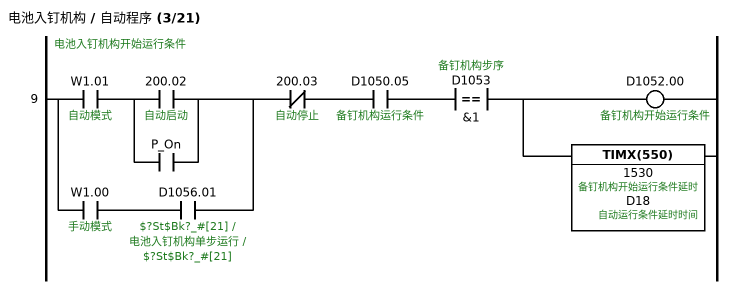
; [picture p96: 电池入钉机构 / 自动程序, rungs 9-9]
; rung 9: 电池入钉机构开始运行条件
LD W1.01  ; 自动模式
LD 200.02  ; 自动启动
OR P_On
ANDLD
LD W1.00  ; 手动模式
AND D1056.01  ; $?St$Bk?_#[21] / 电池入钉机构单步运行 / $?St$Bk?_#[21]
ORLD
ANDNOT 200.03  ; 自动停止
AND D1050.05  ; 备钉机构运行条件
AND=(300) D1053 &1  ; 备钉机构步序
OUT D1052.00  ; 备钉机构开始运行条件
TIMX(550) 1530 D18  ; 自动运行条件延时时间, 备钉机构开始运行条件延时

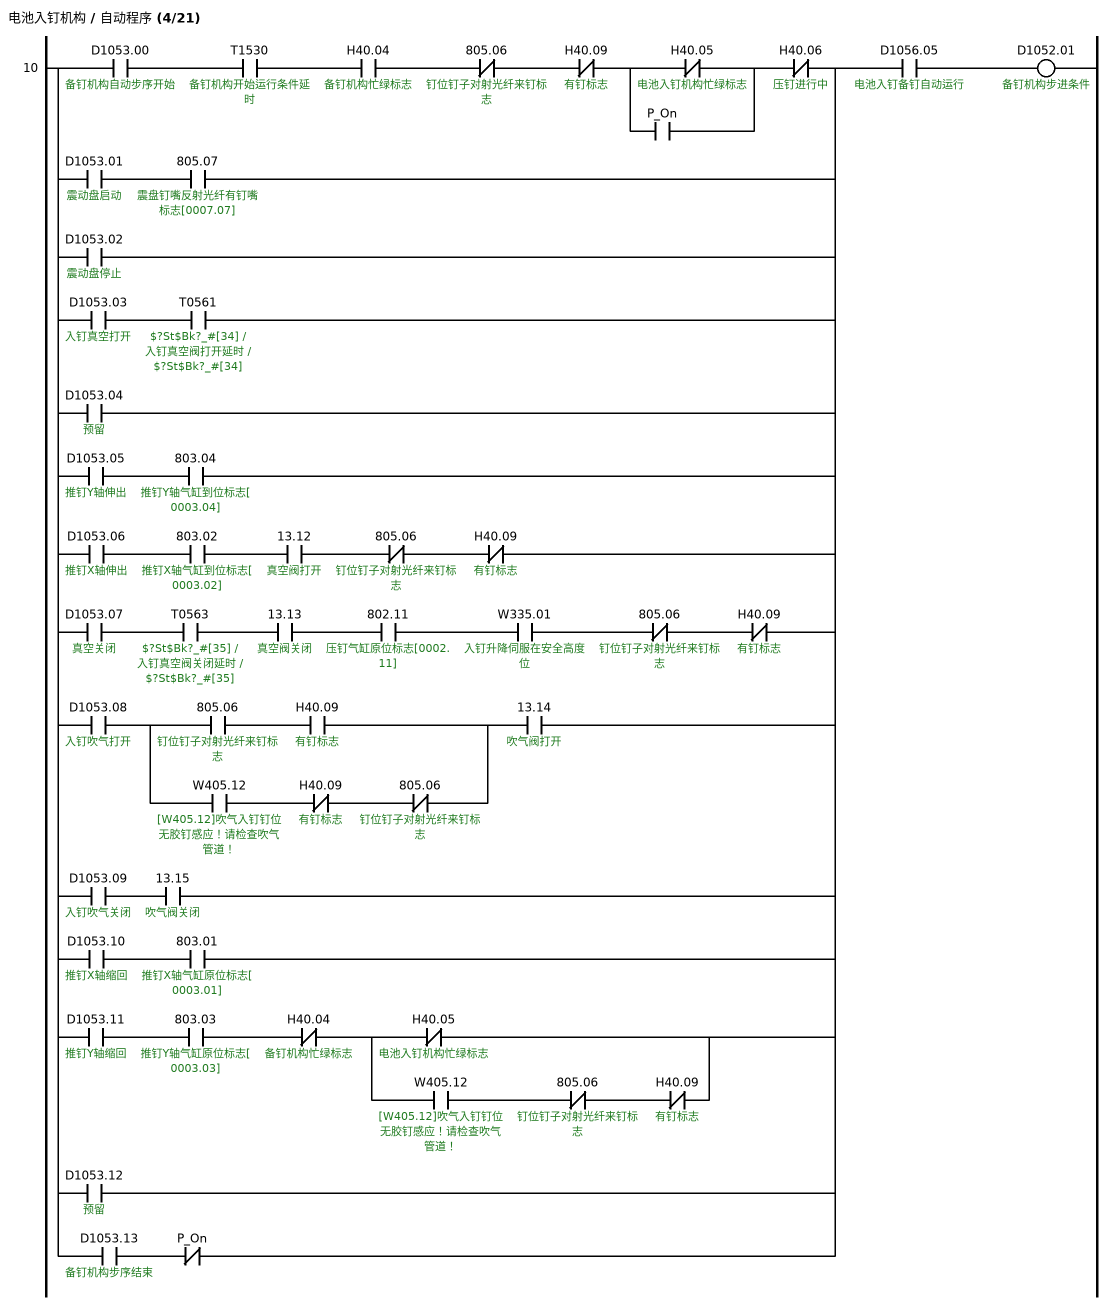
; rung 10
LD D1053.00  ; 备钉机构自动步序开始
AND T1530  ; 备钉机构开始运行条件延时
AND H40.04  ; 备钉机构忙绿标志
ANDNOT 805.06  ; 钉位钉子对射光纤来钉标志
ANDNOT H40.09  ; 有钉标志
LDNOT H40.05  ; 电池入钉机构忙绿标志
OR P_On
ANDLD
ANDNOT H40.06  ; 压钉进行中
LD D1053.01  ; 震动盘启动
AND 805.07  ; 震盘钉嘴反射光纤有钉嘴标志[0007.07]
ORLD
OR D1053.02  ; 震动盘停止
LD D1053.03  ; 入钉真空打开
AND T0561  ; $?St$Bk?_#[34] / 入钉真空阀打开延时 / $?St$Bk?_#[34]
ORLD
OR D1053.04  ; 预留
LD D1053.05  ; 推钉Y轴伸出
AND 803.04  ; 推钉Y轴气缸到位标志[0003.04]
ORLD
LD D1053.06  ; 推钉X轴伸出
AND 803.02  ; 推钉X轴气缸到位标志[0003.02]
AND 13.12  ; 真空阀打开
ANDNOT 805.06  ; 钉位钉子对射光纤来钉标志
ANDNOT H40.09  ; 有钉标志
ORLD
LD D1053.07  ; 真空关闭
AND T0563  ; $?St$Bk?_#[35] / 入钉真空阀关闭延时 / $?St$Bk?_#[35]
AND 13.13  ; 真空阀关闭
AND 802.11  ; 压钉气缸原位标志[0002.11]
AND W335.01  ; 入钉升降伺服在安全高度位
ANDNOT 805.06  ; 钉位钉子对射光纤来钉标志
ANDNOT H40.09  ; 有钉标志
ORLD
LD D1053.08  ; 入钉吹气打开
LD 805.06  ; 钉位钉子对射光纤来钉标志
AND H40.09  ; 有钉标志
LD W405.12  ; [W405.12]吹气入钉钉位无胶钉感应！请检查吹气管道！
ANDNOT H40.09  ; 有钉标志
ANDNOT 805.06  ; 钉位钉子对射光纤来钉标志
ORLD
ANDLD
AND 13.14  ; 吹气阀打开
ORLD
LD D1053.09  ; 入钉吹气关闭
AND 13.15  ; 吹气阀关闭
ORLD
LD D1053.10  ; 推钉X轴缩回
AND 803.01  ; 推钉X轴气缸原位标志[0003.01]
ORLD
LD D1053.11  ; 推钉Y轴缩回
AND 803.03  ; 推钉Y轴气缸原位标志[0003.03]
ANDNOT H40.04  ; 备钉机构忙绿标志
LDNOT H40.05  ; 电池入钉机构忙绿标志
LD W405.12  ; [W405.12]吹气入钉钉位无胶钉感应！请检查吹气管道！
ANDNOT 805.06  ; 钉位钉子对射光纤来钉标志
ANDNOT H40.09  ; 有钉标志
ORLD
ANDLD
ORLD
OR D1053.12  ; 预留
LD D1053.13  ; 备钉机构步序结束
ANDNOT P_On
ORLD
AND D1056.05  ; 电池入钉备钉自动运行
OUT D1052.01  ; 备钉机构步进条件

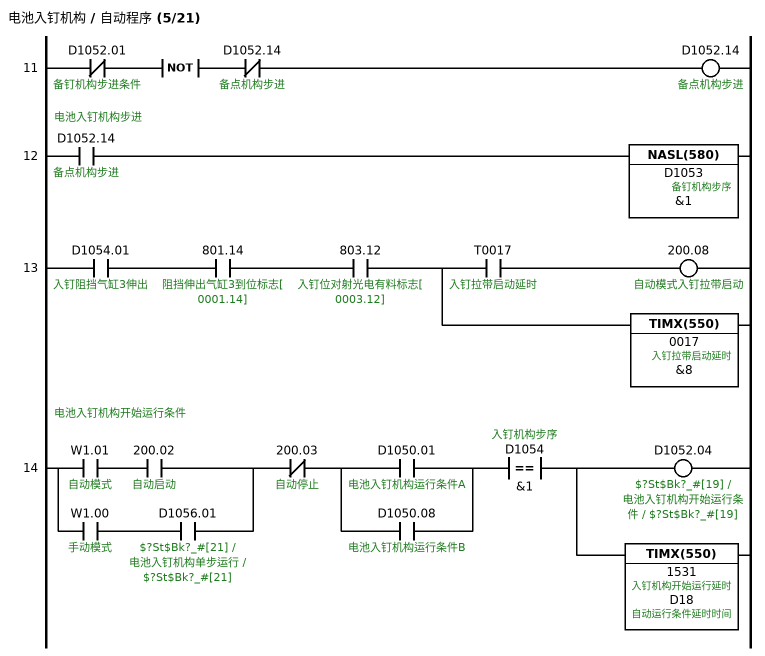
; rung 11
LDNOT D1052.01  ; 备钉机构步进条件
NOT(520)
ANDNOT D1052.14  ; 备点机构步进
OUT D1052.14  ; 备点机构步进
; rung 12: 电池入钉机构步进
LD D1052.14  ; 备点机构步进
NASL(580) D1053 &1  ; 备钉机构步序
; rung 13
LD D1054.01  ; 入钉阻挡气缸3伸出
AND 801.14  ; 阻挡伸出气缸3到位标志[0001.14]
AND 803.12  ; 入钉位对射光电有料标志[0003.12]
OUT TR0
AND T0017  ; 入钉拉带启动延时
OUT 200.08  ; 自动模式入钉拉带启动
LD TR0
TIMX(550) 0017 &8  ; 入钉拉带启动延时
; rung 14: 电池入钉机构开始运行条件
LD W1.01  ; 自动模式
AND 200.02  ; 自动启动
LD W1.00  ; 手动模式
AND D1056.01  ; $?St$Bk?_#[21] / 电池入钉机构单步运行 / $?St$Bk?_#[21]
ORLD
ANDNOT 200.03  ; 自动停止
LD D1050.01  ; 电池入钉机构运行条件A
OR D1050.08  ; 电池入钉机构运行条件B
ANDLD
AND=(300) D1054 &1  ; 入钉机构步序
OUT D1052.04  ; $?St$Bk?_#[19] / 电池入钉机构开始运行条件 / $?St$Bk?_#[19]
TIMX(550) 1531 D18  ; 自动运行条件延时时间, 入钉机构开始运行延时

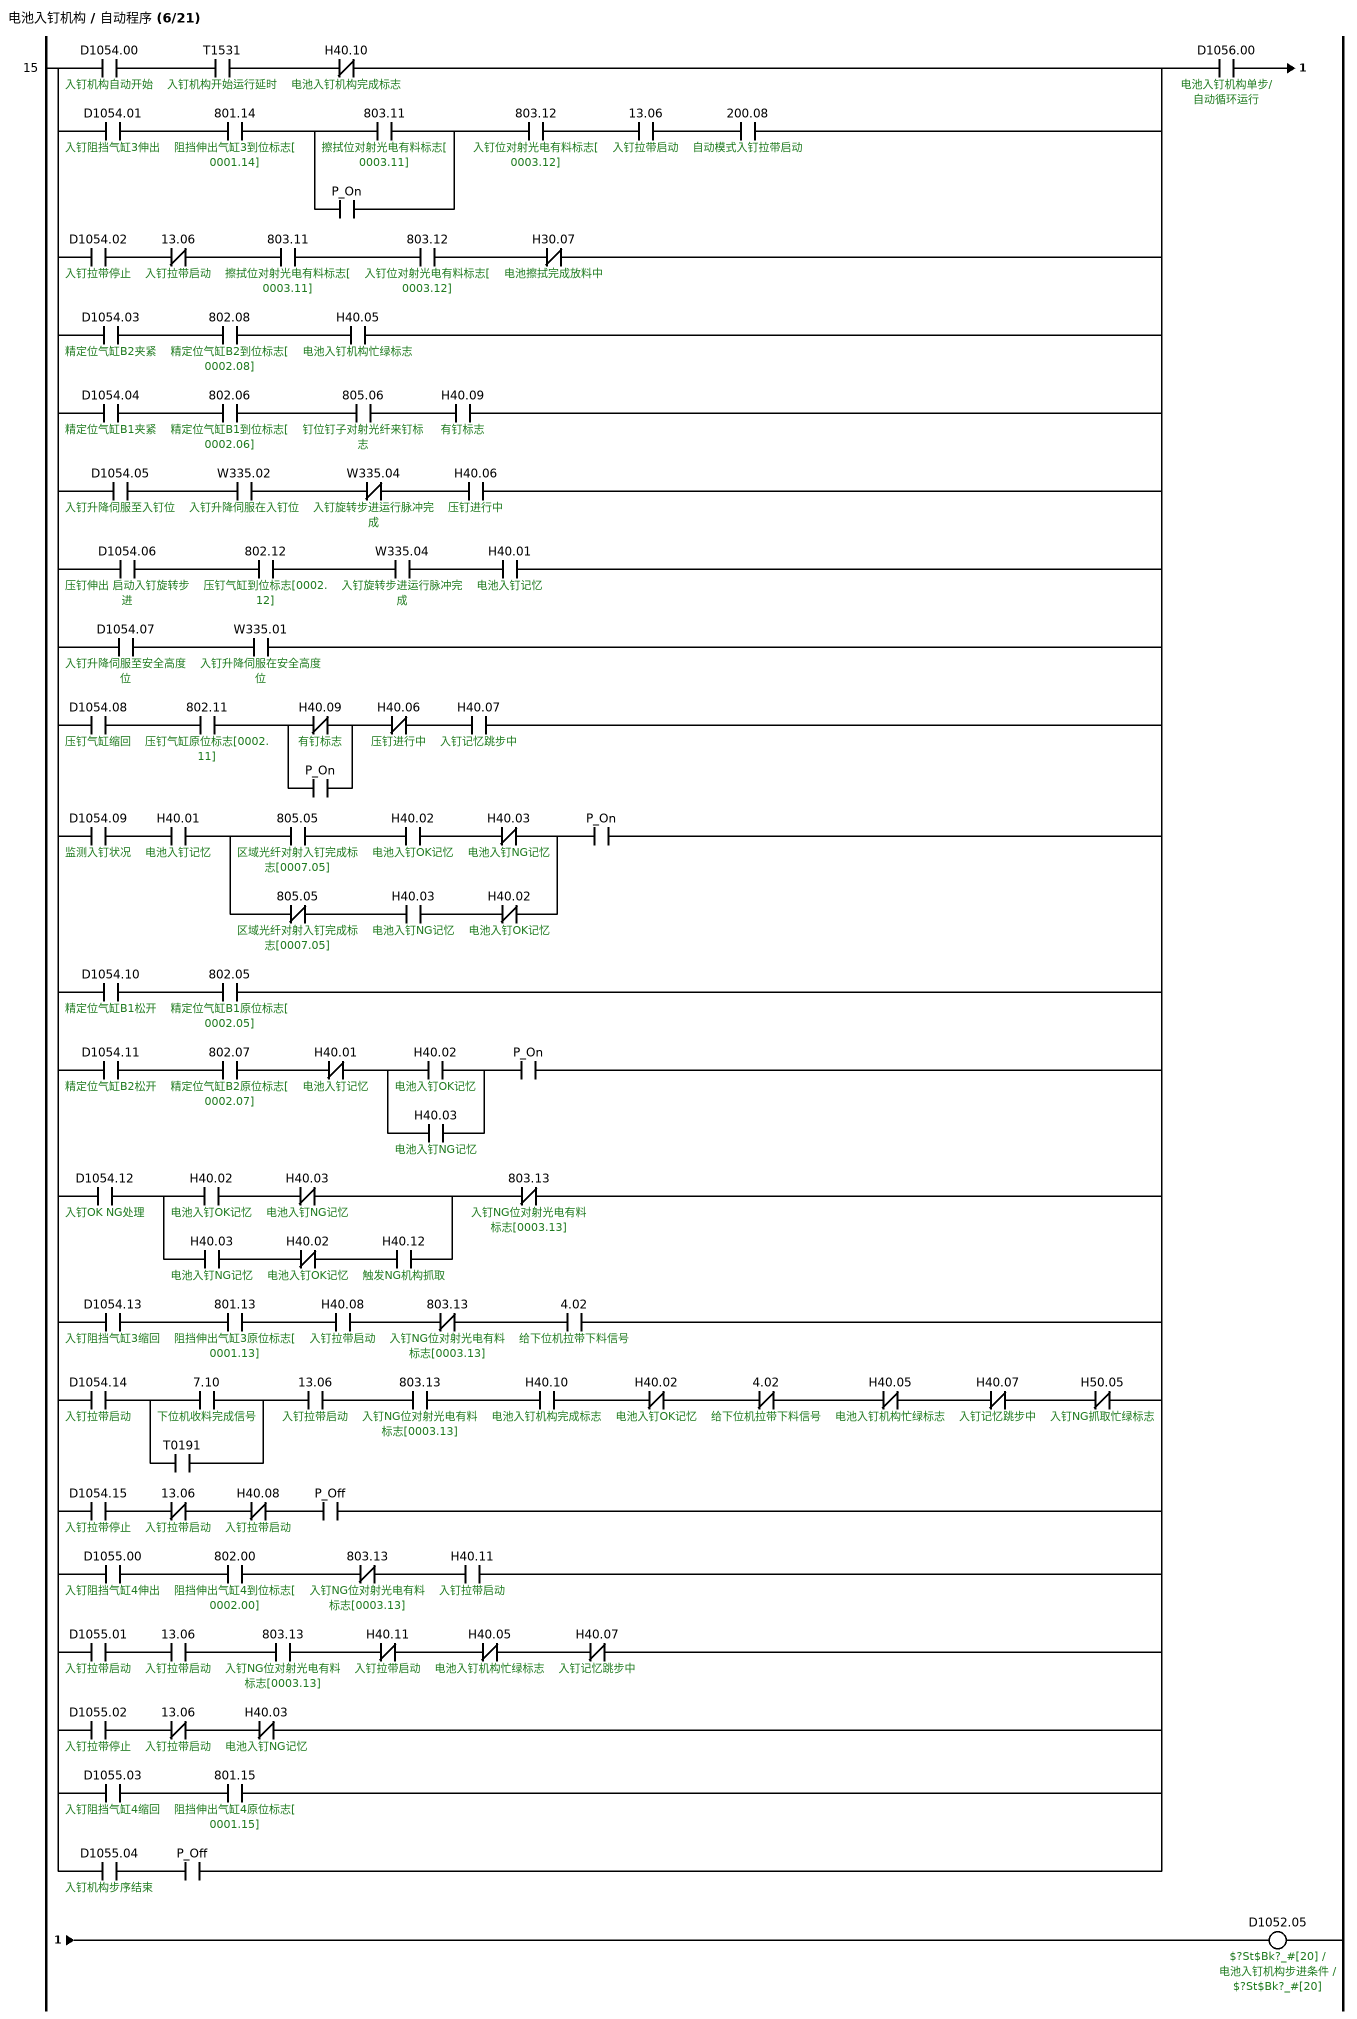
; rung 15
LD D1054.00  ; 入钉机构自动开始
AND T1531  ; 入钉机构开始运行延时
ANDNOT H40.10  ; 电池入钉机构完成标志
LD D1054.01  ; 入钉阻挡气缸3伸出
AND 801.14  ; 阻挡伸出气缸3到位标志[0001.14]
LD 803.11  ; 擦拭位对射光电有料标志[0003.11]
OR P_On
ANDLD
AND 803.12  ; 入钉位对射光电有料标志[0003.12]
AND 13.06  ; 入钉拉带启动
AND 200.08  ; 自动模式入钉拉带启动
ORLD
LD D1054.02  ; 入钉拉带停止
ANDNOT 13.06  ; 入钉拉带启动
AND 803.11  ; 擦拭位对射光电有料标志[0003.11]
AND 803.12  ; 入钉位对射光电有料标志[0003.12]
ANDNOT H30.07  ; 电池擦拭完成放料中
ORLD
LD D1054.03  ; 精定位气缸B2夹紧
AND 802.08  ; 精定位气缸B2到位标志[0002.08]
AND H40.05  ; 电池入钉机构忙绿标志
ORLD
LD D1054.04  ; 精定位气缸B1夹紧
AND 802.06  ; 精定位气缸B1到位标志[0002.06]
AND 805.06  ; 钉位钉子对射光纤来钉标志
AND H40.09  ; 有钉标志
ORLD
LD D1054.05  ; 入钉升降伺服至入钉位
AND W335.02  ; 入钉升降伺服在入钉位
ANDNOT W335.04  ; 入钉旋转步进运行脉冲完成
AND H40.06  ; 压钉进行中
ORLD
LD D1054.06  ; 压钉伸出 启动入钉旋转步进
AND 802.12  ; 压钉气缸到位标志[0002.12]
AND W335.04  ; 入钉旋转步进运行脉冲完成
AND H40.01  ; 电池入钉记忆
ORLD
LD D1054.07  ; 入钉升降伺服至安全高度位
AND W335.01  ; 入钉升降伺服在安全高度位
ORLD
LD D1054.08  ; 压钉气缸缩回
AND 802.11  ; 压钉气缸原位标志[0002.11]
LDNOT H40.09  ; 有钉标志
OR P_On
ANDLD
ANDNOT H40.06  ; 压钉进行中
AND H40.07  ; 入钉记忆跳步中
ORLD
LD D1054.09  ; 监测入钉状况
AND H40.01  ; 电池入钉记忆
LD 805.05  ; 区域光纤对射入钉完成标志[0007.05]
AND H40.02  ; 电池入钉OK记忆
ANDNOT H40.03  ; 电池入钉NG记忆
LDNOT 805.05  ; 区域光纤对射入钉完成标志[0007.05]
AND H40.03  ; 电池入钉NG记忆
ANDNOT H40.02  ; 电池入钉OK记忆
ORLD
ANDLD
AND P_On
ORLD
LD D1054.10  ; 精定位气缸B1松开
AND 802.05  ; 精定位气缸B1原位标志[0002.05]
ORLD
LD D1054.11  ; 精定位气缸B2松开
AND 802.07  ; 精定位气缸B2原位标志[0002.07]
ANDNOT H40.01  ; 电池入钉记忆
LD H40.02  ; 电池入钉OK记忆
OR H40.03  ; 电池入钉NG记忆
ANDLD
AND P_On
ORLD
LD D1054.12  ; 入钉OK NG处理
LD H40.02  ; 电池入钉OK记忆
ANDNOT H40.03  ; 电池入钉NG记忆
LD H40.03  ; 电池入钉NG记忆
ANDNOT H40.02  ; 电池入钉OK记忆
AND H40.12  ; 触发NG机构抓取
ORLD
ANDLD
ANDNOT 803.13  ; 入钉NG位对射光电有料标志[0003.13]
ORLD
LD D1054.13  ; 入钉阻挡气缸3缩回
AND 801.13  ; 阻挡伸出气缸3原位标志[0001.13]
AND H40.08  ; 入钉拉带启动
ANDNOT 803.13  ; 入钉NG位对射光电有料标志[0003.13]
AND 4.02  ; 给下位机拉带下料信号
ORLD
LD D1054.14  ; 入钉拉带启动
LD 7.10  ; 下位机收料完成信号
OR T0191
ANDLD
AND 13.06  ; 入钉拉带启动
AND 803.13  ; 入钉NG位对射光电有料标志[0003.13]
AND H40.10  ; 电池入钉机构完成标志
ANDNOT H40.02  ; 电池入钉OK记忆
ANDNOT 4.02  ; 给下位机拉带下料信号
ANDNOT H40.05  ; 电池入钉机构忙绿标志
ANDNOT H40.07  ; 入钉记忆跳步中
ANDNOT H50.05  ; 入钉NG抓取忙绿标志
ORLD
LD D1054.15  ; 入钉拉带停止
ANDNOT 13.06  ; 入钉拉带启动
ANDNOT H40.08  ; 入钉拉带启动
AND P_Off
ORLD
LD D1055.00  ; 入钉阻挡气缸4伸出
AND 802.00  ; 阻挡伸出气缸4到位标志[0002.00]
ANDNOT 803.13  ; 入钉NG位对射光电有料标志[0003.13]
AND H40.11  ; 入钉拉带启动
ORLD
LD D1055.01  ; 入钉拉带启动
AND 13.06  ; 入钉拉带启动
AND 803.13  ; 入钉NG位对射光电有料标志[0003.13]
ANDNOT H40.11  ; 入钉拉带启动
ANDNOT H40.05  ; 电池入钉机构忙绿标志
ANDNOT H40.07  ; 入钉记忆跳步中
ORLD
LD D1055.02  ; 入钉拉带停止
ANDNOT 13.06  ; 入钉拉带启动
ANDNOT H40.03  ; 电池入钉NG记忆
ORLD
LD D1055.03  ; 入钉阻挡气缸4缩回
AND 801.15  ; 阻挡伸出气缸4原位标志[0001.15]
ORLD
LD D1055.04  ; 入钉机构步序结束
AND P_Off
ORLD
AND D1056.00  ; 电池入钉机构单步/自动循环运行
OUT D1052.05  ; $?St$Bk?_#[20] / 电池入钉机构步进条件 / $?St$Bk?_#[20]

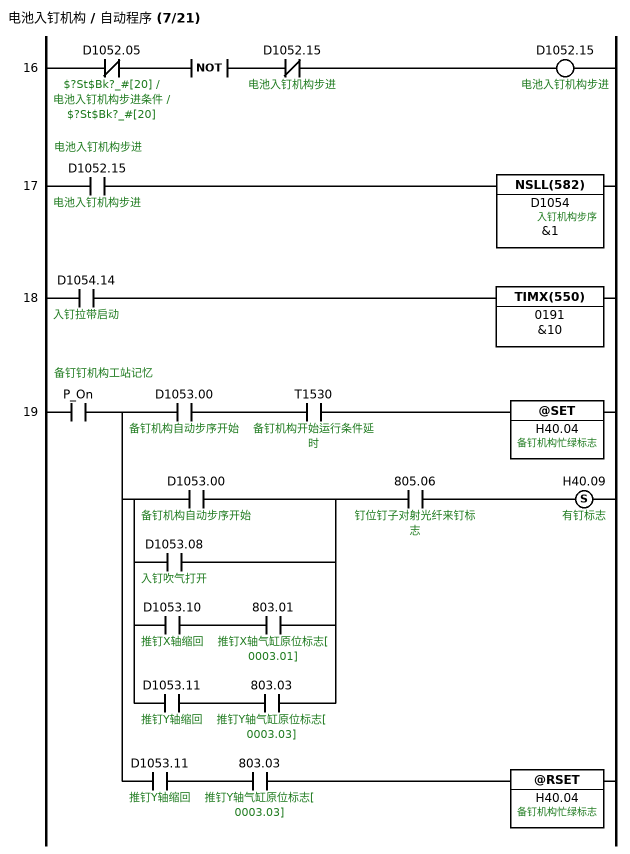
; rung 16
LDNOT D1052.05  ; $?St$Bk?_#[20] / 电池入钉机构步进条件 / $?St$Bk?_#[20]
NOT(520)
ANDNOT D1052.15  ; 电池入钉机构步进
OUT D1052.15  ; 电池入钉机构步进
; rung 17: 电池入钉机构步进
LD D1052.15  ; 电池入钉机构步进
NSLL(582) D1054 &1  ; 入钉机构步序
; rung 18
LD D1054.14  ; 入钉拉带启动
TIMX(550) 0191 &10
; rung 19: 备钉钉机构工站记忆
LD P_On
OUT TR0
AND D1053.00  ; 备钉机构自动步序开始
AND T1530  ; 备钉机构开始运行条件延时
@SET H40.04  ; 备钉机构忙绿标志
LD TR0
LD D1053.00  ; 备钉机构自动步序开始
OR D1053.08  ; 入钉吹气打开
LD D1053.10  ; 推钉X轴缩回
AND 803.01  ; 推钉X轴气缸原位标志[0003.01]
ORLD
LD D1053.11  ; 推钉Y轴缩回
AND 803.03  ; 推钉Y轴气缸原位标志[0003.03]
ORLD
ANDLD
AND 805.06  ; 钉位钉子对射光纤来钉标志
SET H40.09  ; 有钉标志
LD TR0
AND D1053.11  ; 推钉Y轴缩回
AND 803.03  ; 推钉Y轴气缸原位标志[0003.03]
@RSET H40.04  ; 备钉机构忙绿标志

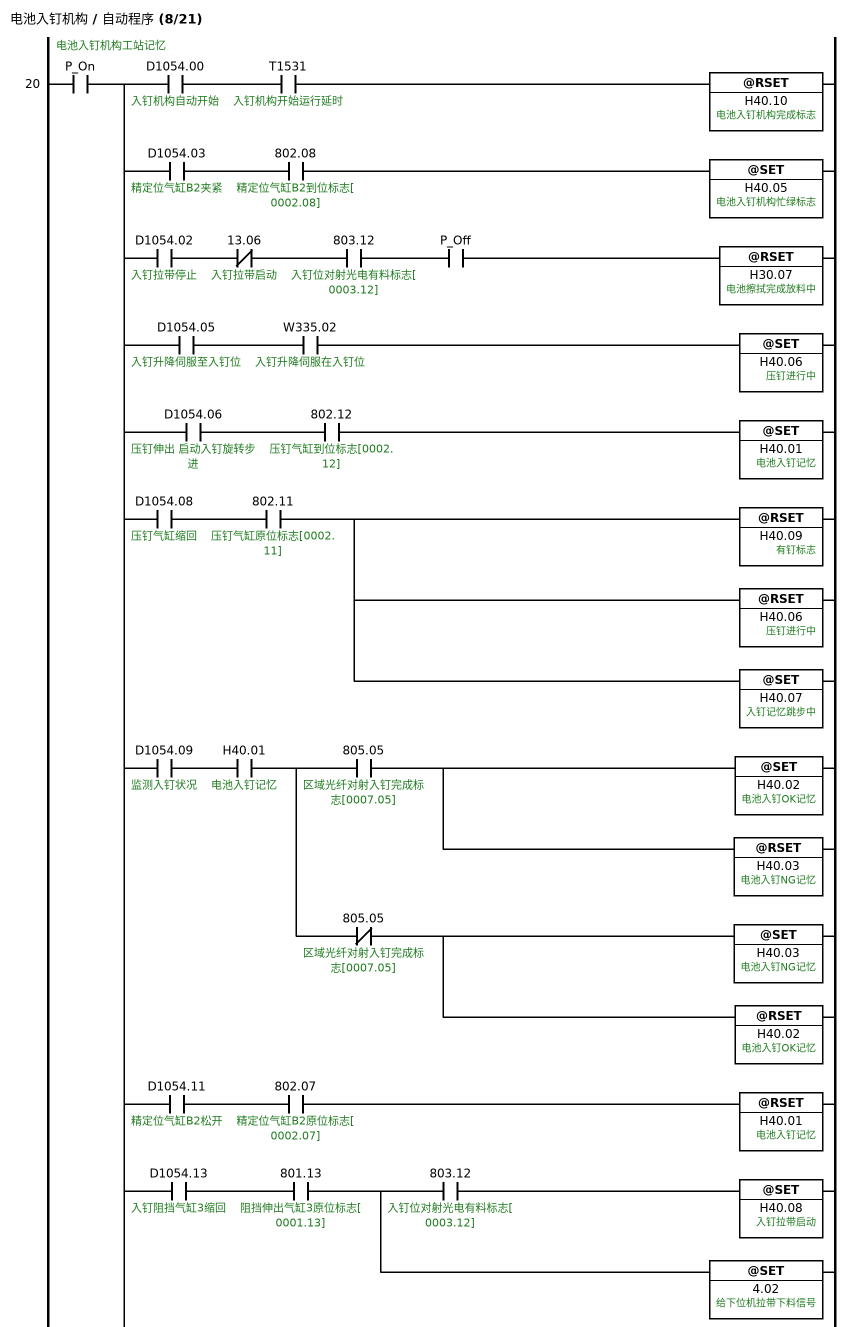

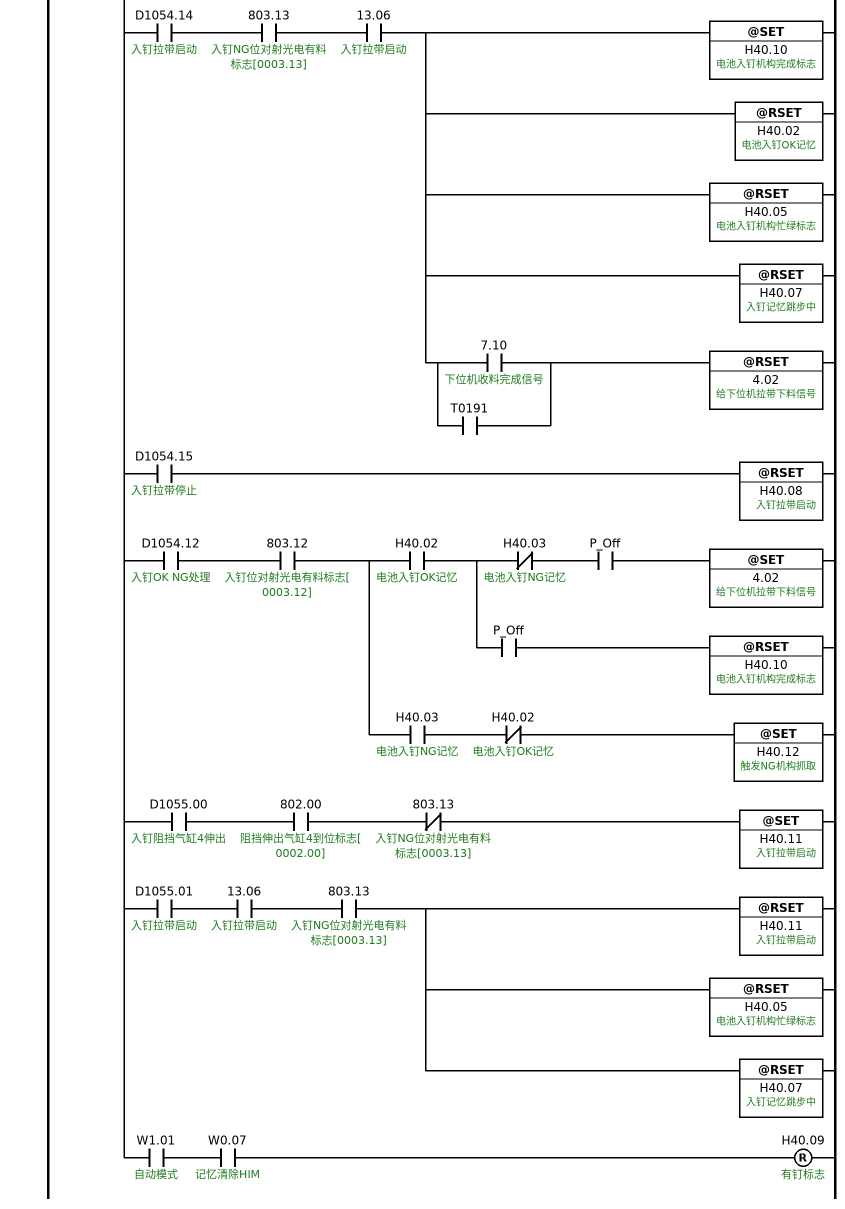
; rung 20: 电池入钉机构工站记忆
LD P_On
OUT TR0
AND D1054.00  ; 入钉机构自动开始
AND T1531  ; 入钉机构开始运行延时
@RSET H40.10  ; 电池入钉机构完成标志
LD TR0
AND D1054.03  ; 精定位气缸B2夹紧
AND 802.08  ; 精定位气缸B2到位标志[0002.08]
@SET H40.05  ; 电池入钉机构忙绿标志
LD TR0
AND D1054.02  ; 入钉拉带停止
ANDNOT 13.06  ; 入钉拉带启动
AND 803.12  ; 入钉位对射光电有料标志[0003.12]
AND P_Off
@RSET H30.07  ; 电池擦拭完成放料中
LD TR0
AND D1054.05  ; 入钉升降伺服至入钉位
AND W335.02  ; 入钉升降伺服在入钉位
@SET H40.06  ; 压钉进行中
LD TR0
AND D1054.06  ; 压钉伸出 启动入钉旋转步进
AND 802.12  ; 压钉气缸到位标志[0002.12]
@SET H40.01  ; 电池入钉记忆
LD TR0
AND D1054.08  ; 压钉气缸缩回
AND 802.11  ; 压钉气缸原位标志[0002.11]
@RSET H40.09  ; 有钉标志
@RSET H40.06  ; 压钉进行中
@SET H40.07  ; 入钉记忆跳步中
LD TR0
AND D1054.09  ; 监测入钉状况
AND H40.01  ; 电池入钉记忆
OUT TR1
AND 805.05  ; 区域光纤对射入钉完成标志[0007.05]
@SET H40.02  ; 电池入钉OK记忆
@RSET H40.03  ; 电池入钉NG记忆
LD TR1
ANDNOT 805.05  ; 区域光纤对射入钉完成标志[0007.05]
@SET H40.03  ; 电池入钉NG记忆
@RSET H40.02  ; 电池入钉OK记忆
LD TR0
AND D1054.11  ; 精定位气缸B2松开
AND 802.07  ; 精定位气缸B2原位标志[0002.07]
@RSET H40.01  ; 电池入钉记忆
LD TR0
AND D1054.13  ; 入钉阻挡气缸3缩回
AND 801.13  ; 阻挡伸出气缸3原位标志[0001.13]
OUT TR1
AND 803.12  ; 入钉位对射光电有料标志[0003.12]
@SET H40.08  ; 入钉拉带启动
LD TR1
@SET 4.02  ; 给下位机拉带下料信号
LD TR0
AND D1054.14  ; 入钉拉带启动
AND 803.13  ; 入钉NG位对射光电有料标志[0003.13]
AND 13.06  ; 入钉拉带启动
@SET H40.10  ; 电池入钉机构完成标志
@RSET H40.02  ; 电池入钉OK记忆
@RSET H40.05  ; 电池入钉机构忙绿标志
@RSET H40.07  ; 入钉记忆跳步中
LD 7.10  ; 下位机收料完成信号
OR T0191
ANDLD
@RSET 4.02  ; 给下位机拉带下料信号
LD TR0
AND D1054.15  ; 入钉拉带停止
@RSET H40.08  ; 入钉拉带启动
LD TR0
AND D1054.12  ; 入钉OK NG处理
AND 803.12  ; 入钉位对射光电有料标志[0003.12]
OUT TR1
AND H40.02  ; 电池入钉OK记忆
OUT TR2
ANDNOT H40.03  ; 电池入钉NG记忆
AND P_Off
@SET 4.02  ; 给下位机拉带下料信号
LD TR2
AND P_Off
@RSET H40.10  ; 电池入钉机构完成标志
LD TR1
AND H40.03  ; 电池入钉NG记忆
ANDNOT H40.02  ; 电池入钉OK记忆
@SET H40.12  ; 触发NG机构抓取
LD TR0
AND D1055.00  ; 入钉阻挡气缸4伸出
AND 802.00  ; 阻挡伸出气缸4到位标志[0002.00]
ANDNOT 803.13  ; 入钉NG位对射光电有料标志[0003.13]
@SET H40.11  ; 入钉拉带启动
LD TR0
AND D1055.01  ; 入钉拉带启动
AND 13.06  ; 入钉拉带启动
AND 803.13  ; 入钉NG位对射光电有料标志[0003.13]
@RSET H40.11  ; 入钉拉带启动
@RSET H40.05  ; 电池入钉机构忙绿标志
@RSET H40.07  ; 入钉记忆跳步中
LD TR0
AND W1.01  ; 自动模式
AND W0.07  ; 记忆清除HIM
RSET H40.09  ; 有钉标志

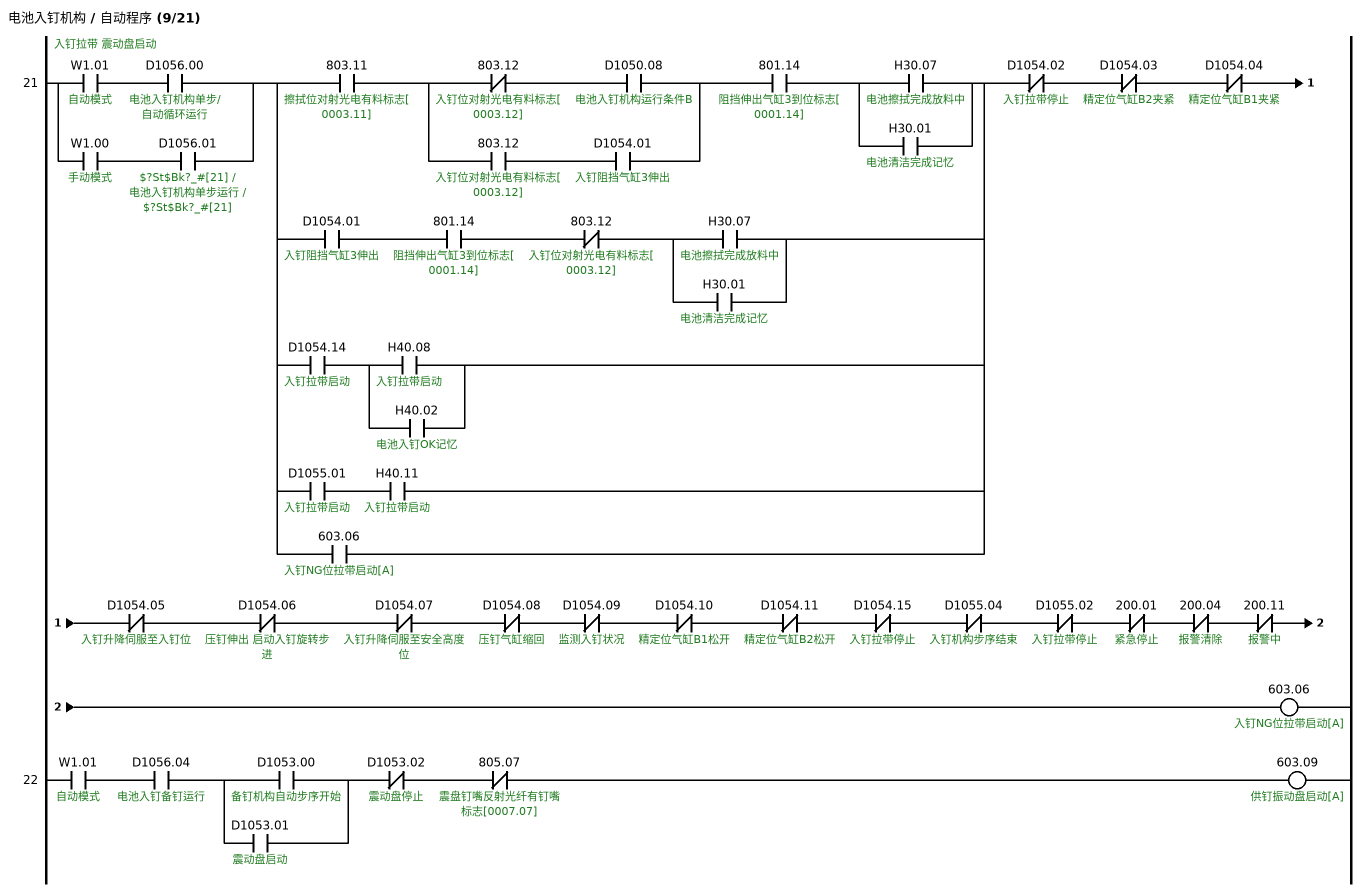
; rung 21: 入钉拉带 震动盘启动
LD W1.01  ; 自动模式
AND D1056.00  ; 电池入钉机构单步/自动循环运行
LD W1.00  ; 手动模式
AND D1056.01  ; $?St$Bk?_#[21] / 电池入钉机构单步运行 / $?St$Bk?_#[21]
ORLD
LD 803.11  ; 擦拭位对射光电有料标志[0003.11]
LDNOT 803.12  ; 入钉位对射光电有料标志[0003.12]
AND D1050.08  ; 电池入钉机构运行条件B
LD 803.12  ; 入钉位对射光电有料标志[0003.12]
AND D1054.01  ; 入钉阻挡气缸3伸出
ORLD
ANDLD
AND 801.14  ; 阻挡伸出气缸3到位标志[0001.14]
LD H30.07  ; 电池擦拭完成放料中
OR H30.01  ; 电池清洁完成记忆
ANDLD
LD D1054.01  ; 入钉阻挡气缸3伸出
AND 801.14  ; 阻挡伸出气缸3到位标志[0001.14]
ANDNOT 803.12  ; 入钉位对射光电有料标志[0003.12]
LD H30.07  ; 电池擦拭完成放料中
OR H30.01  ; 电池清洁完成记忆
ANDLD
ORLD
LD D1054.14  ; 入钉拉带启动
LD H40.08  ; 入钉拉带启动
OR H40.02  ; 电池入钉OK记忆
ANDLD
ORLD
LD D1055.01  ; 入钉拉带启动
AND H40.11  ; 入钉拉带启动
ORLD
OR 603.06  ; 入钉NG位拉带启动[A]
ANDLD
ANDNOT D1054.02  ; 入钉拉带停止
ANDNOT D1054.03  ; 精定位气缸B2夹紧
ANDNOT D1054.04  ; 精定位气缸B1夹紧
ANDNOT D1054.05  ; 入钉升降伺服至入钉位
ANDNOT D1054.06  ; 压钉伸出 启动入钉旋转步进
ANDNOT D1054.07  ; 入钉升降伺服至安全高度位
ANDNOT D1054.08  ; 压钉气缸缩回
ANDNOT D1054.09  ; 监测入钉状况
ANDNOT D1054.10  ; 精定位气缸B1松开
ANDNOT D1054.11  ; 精定位气缸B2松开
ANDNOT D1054.15  ; 入钉拉带停止
ANDNOT D1055.04  ; 入钉机构步序结束
ANDNOT D1055.02  ; 入钉拉带停止
ANDNOT 200.01  ; 紧急停止
ANDNOT 200.04  ; 报警清除
ANDNOT 200.11  ; 报警中
OUT 603.06  ; 入钉NG位拉带启动[A]
; rung 22
LD W1.01  ; 自动模式
AND D1056.04  ; 电池入钉备钉运行
LD D1053.00  ; 备钉机构自动步序开始
OR D1053.01  ; 震动盘启动
ANDLD
ANDNOT D1053.02  ; 震动盘停止
ANDNOT 805.07  ; 震盘钉嘴反射光纤有钉嘴标志[0007.07]
OUT 603.09  ; 供钉振动盘启动[A]

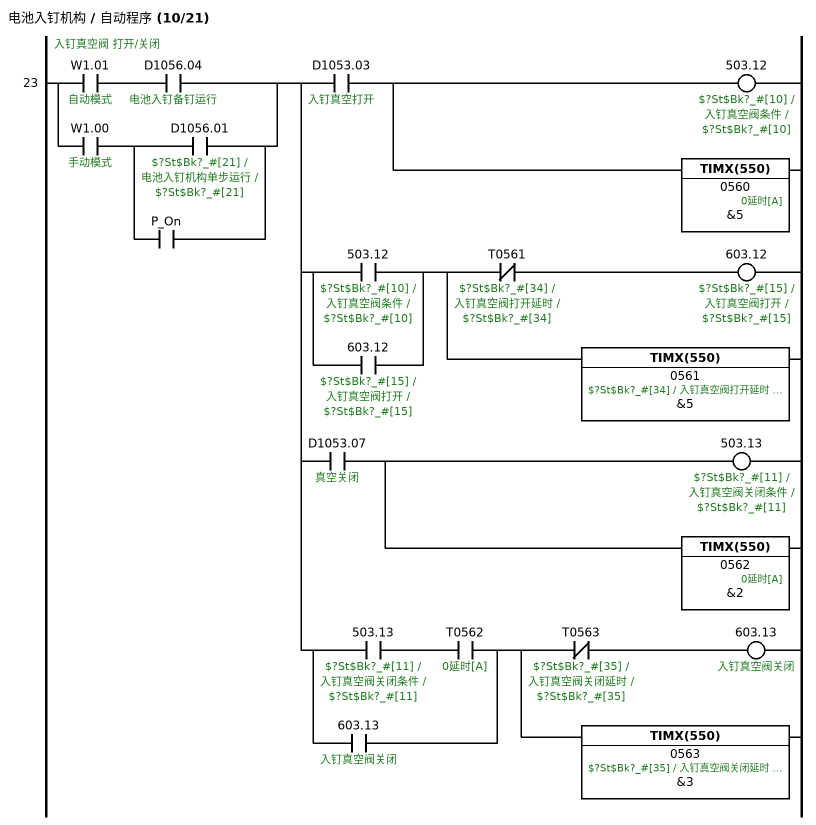
; rung 23: 入钉真空阀 打开/关闭
LD W1.01  ; 自动模式
AND D1056.04  ; 电池入钉备钉运行
LD W1.00  ; 手动模式
LD D1056.01  ; $?St$Bk?_#[21] / 电池入钉机构单步运行 / $?St$Bk?_#[21]
OR P_On
ANDLD
ORLD
OUT TR0
AND D1053.03  ; 入钉真空打开
OUT 503.12  ; $?St$Bk?_#[10] / 入钉真空阀条件 / $?St$Bk?_#[10]
TIMX(550) 0560 &5  ; 0延时[A]
LD TR0
LD 503.12  ; $?St$Bk?_#[10] / 入钉真空阀条件 / $?St$Bk?_#[10]
OR 603.12  ; $?St$Bk?_#[15] / 入钉真空阀打开 / $?St$Bk?_#[15]
ANDLD
OUT TR1
ANDNOT T0561  ; $?St$Bk?_#[34] / 入钉真空阀打开延时 / $?St$Bk?_#[34]
OUT 603.12  ; $?St$Bk?_#[15] / 入钉真空阀打开 / $?St$Bk?_#[15]
LD TR1
TIMX(550) 0561 &5  ; $?St$Bk?_#[34] / 入钉真空阀打开延时 / $?St$Bk?_#[34]
LD TR0
AND D1053.07  ; 真空关闭
OUT 503.13  ; $?St$Bk?_#[11] / 入钉真空阀关闭条件 / $?St$Bk?_#[11]
TIMX(550) 0562 &2  ; 0延时[A]
LD TR0
LD 503.13  ; $?St$Bk?_#[11] / 入钉真空阀关闭条件 / $?St$Bk?_#[11]
AND T0562  ; 0延时[A]
OR 603.13  ; 入钉真空阀关闭
ANDLD
OUT TR0
ANDNOT T0563  ; $?St$Bk?_#[35] / 入钉真空阀关闭延时 / $?St$Bk?_#[35]
OUT 603.13  ; 入钉真空阀关闭
LD TR0
TIMX(550) 0563 &3  ; $?St$Bk?_#[35] / 入钉真空阀关闭延时 / $?St$Bk?_#[35]

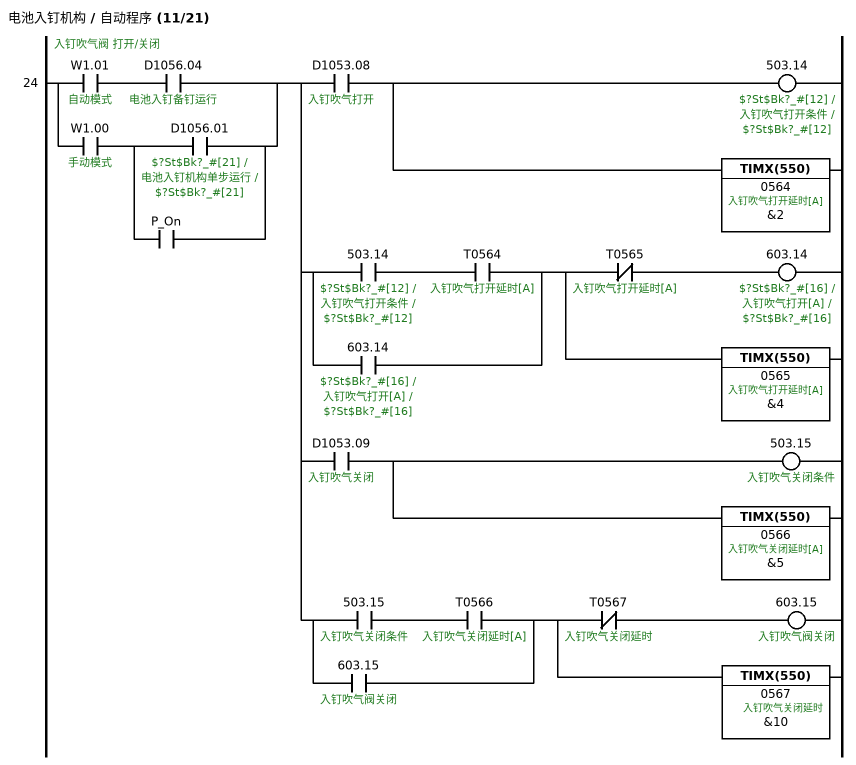
; rung 24: 入钉吹气阀 打开/关闭
LD W1.01  ; 自动模式
AND D1056.04  ; 电池入钉备钉运行
LD W1.00  ; 手动模式
LD D1056.01  ; $?St$Bk?_#[21] / 电池入钉机构单步运行 / $?St$Bk?_#[21]
OR P_On
ANDLD
ORLD
OUT TR0
AND D1053.08  ; 入钉吹气打开
OUT 503.14  ; $?St$Bk?_#[12] / 入钉吹气打开条件 / $?St$Bk?_#[12]
TIMX(550) 0564 &2  ; 入钉吹气打开延时[A]
LD TR0
LD 503.14  ; $?St$Bk?_#[12] / 入钉吹气打开条件 / $?St$Bk?_#[12]
AND T0564  ; 入钉吹气打开延时[A]
OR 603.14  ; $?St$Bk?_#[16] / 入钉吹气打开[A] / $?St$Bk?_#[16]
ANDLD
OUT TR1
ANDNOT T0565  ; 入钉吹气打开延时[A]
OUT 603.14  ; $?St$Bk?_#[16] / 入钉吹气打开[A] / $?St$Bk?_#[16]
LD TR1
TIMX(550) 0565 &4  ; 入钉吹气打开延时[A]
LD TR0
AND D1053.09  ; 入钉吹气关闭
OUT 503.15  ; 入钉吹气关闭条件
TIMX(550) 0566 &5  ; 入钉吹气关闭延时[A]
LD TR0
LD 503.15  ; 入钉吹气关闭条件
AND T0566  ; 入钉吹气关闭延时[A]
OR 603.15  ; 入钉吹气阀关闭
ANDLD
OUT TR0
ANDNOT T0567  ; 入钉吹气关闭延时
OUT 603.15  ; 入钉吹气阀关闭
LD TR0
TIMX(550) 0567 &10  ; 入钉吹气关闭延时

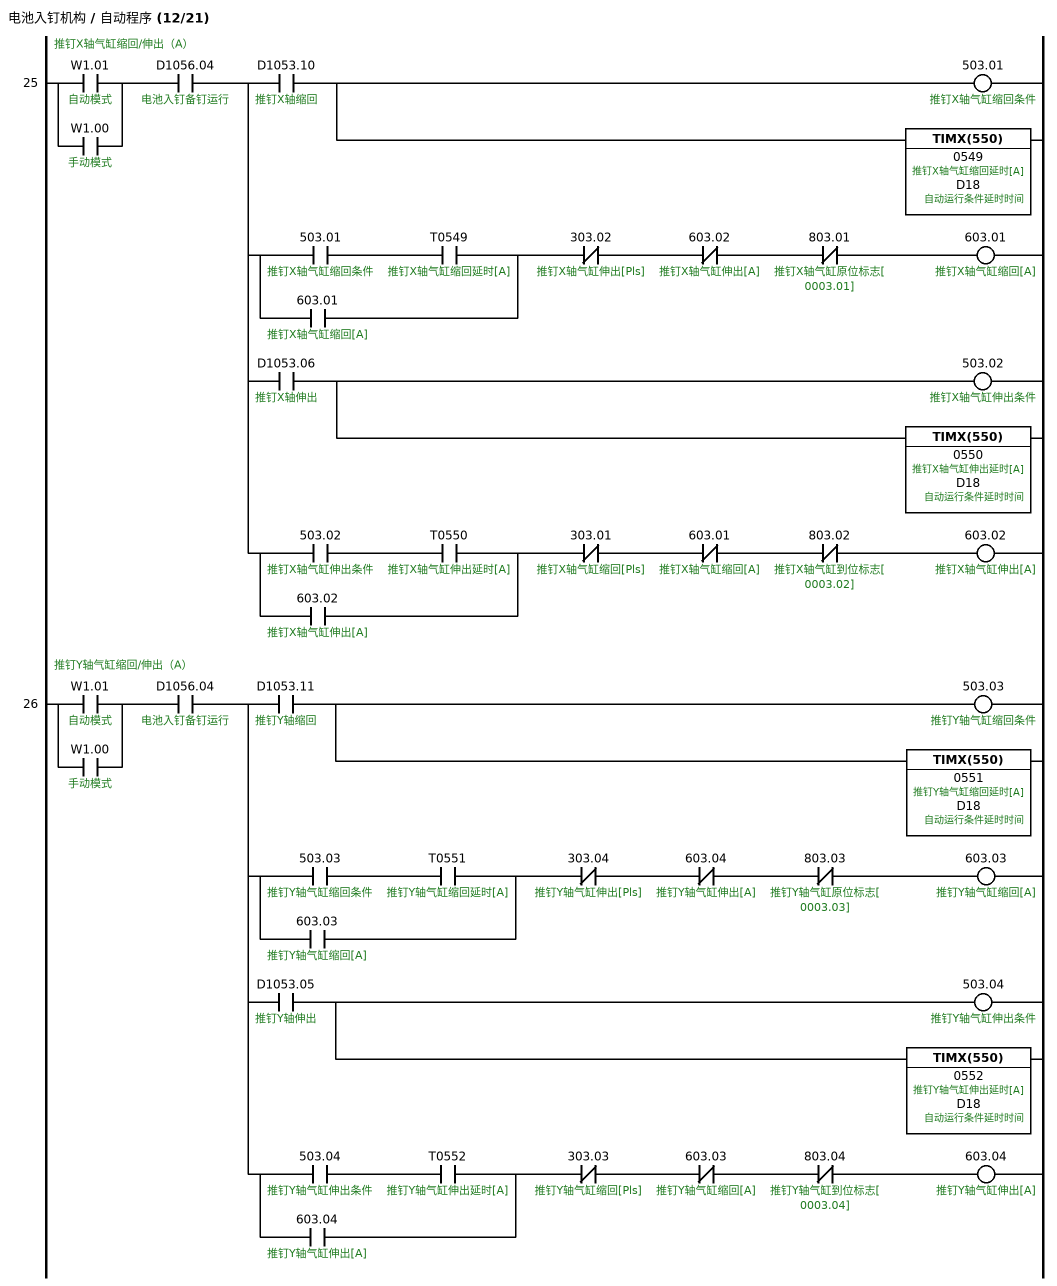
; rung 25: 推钉X轴气缸缩回/伸出（A）
LD W1.01  ; 自动模式
OR W1.00  ; 手动模式
AND D1056.04  ; 电池入钉备钉运行
OUT TR0
AND D1053.10  ; 推钉X轴缩回
OUT 503.01  ; 推钉X轴气缸缩回条件
TIMX(550) 0549 D18  ; 自动运行条件延时时间, 推钉X轴气缸缩回延时[A]
LD TR0
LD 503.01  ; 推钉X轴气缸缩回条件
AND T0549  ; 推钉X轴气缸缩回延时[A]
OR 603.01  ; 推钉X轴气缸缩回[A]
ANDLD
ANDNOT 303.02  ; 推钉X轴气缸伸出[Pls]
ANDNOT 603.02  ; 推钉X轴气缸伸出[A]
ANDNOT 803.01  ; 推钉X轴气缸原位标志[0003.01]
OUT 603.01  ; 推钉X轴气缸缩回[A]
LD TR0
AND D1053.06  ; 推钉X轴伸出
OUT 503.02  ; 推钉X轴气缸伸出条件
TIMX(550) 0550 D18  ; 自动运行条件延时时间, 推钉X轴气缸伸出延时[A]
LD TR0
LD 503.02  ; 推钉X轴气缸伸出条件
AND T0550  ; 推钉X轴气缸伸出延时[A]
OR 603.02  ; 推钉X轴气缸伸出[A]
ANDLD
ANDNOT 303.01  ; 推钉X轴气缸缩回[Pls]
ANDNOT 603.01  ; 推钉X轴气缸缩回[A]
ANDNOT 803.02  ; 推钉X轴气缸到位标志[0003.02]
OUT 603.02  ; 推钉X轴气缸伸出[A]
; rung 26: 推钉Y轴气缸缩回/伸出（A）
LD W1.01  ; 自动模式
OR W1.00  ; 手动模式
AND D1056.04  ; 电池入钉备钉运行
OUT TR0
AND D1053.11  ; 推钉Y轴缩回
OUT 503.03  ; 推钉Y轴气缸缩回条件
TIMX(550) 0551 D18  ; 自动运行条件延时时间, 推钉Y轴气缸缩回延时[A]
LD TR0
LD 503.03  ; 推钉Y轴气缸缩回条件
AND T0551  ; 推钉Y轴气缸缩回延时[A]
OR 603.03  ; 推钉Y轴气缸缩回[A]
ANDLD
ANDNOT 303.04  ; 推钉Y轴气缸伸出[Pls]
ANDNOT 603.04  ; 推钉Y轴气缸伸出[A]
ANDNOT 803.03  ; 推钉Y轴气缸原位标志[0003.03]
OUT 603.03  ; 推钉Y轴气缸缩回[A]
LD TR0
AND D1053.05  ; 推钉Y轴伸出
OUT 503.04  ; 推钉Y轴气缸伸出条件
TIMX(550) 0552 D18  ; 自动运行条件延时时间, 推钉Y轴气缸伸出延时[A]
LD TR0
LD 503.04  ; 推钉Y轴气缸伸出条件
AND T0552  ; 推钉Y轴气缸伸出延时[A]
OR 603.04  ; 推钉Y轴气缸伸出[A]
ANDLD
ANDNOT 303.03  ; 推钉Y轴气缸缩回[Pls]
ANDNOT 603.03  ; 推钉Y轴气缸缩回[A]
ANDNOT 803.04  ; 推钉Y轴气缸到位标志[0003.04]
OUT 603.04  ; 推钉Y轴气缸伸出[A]

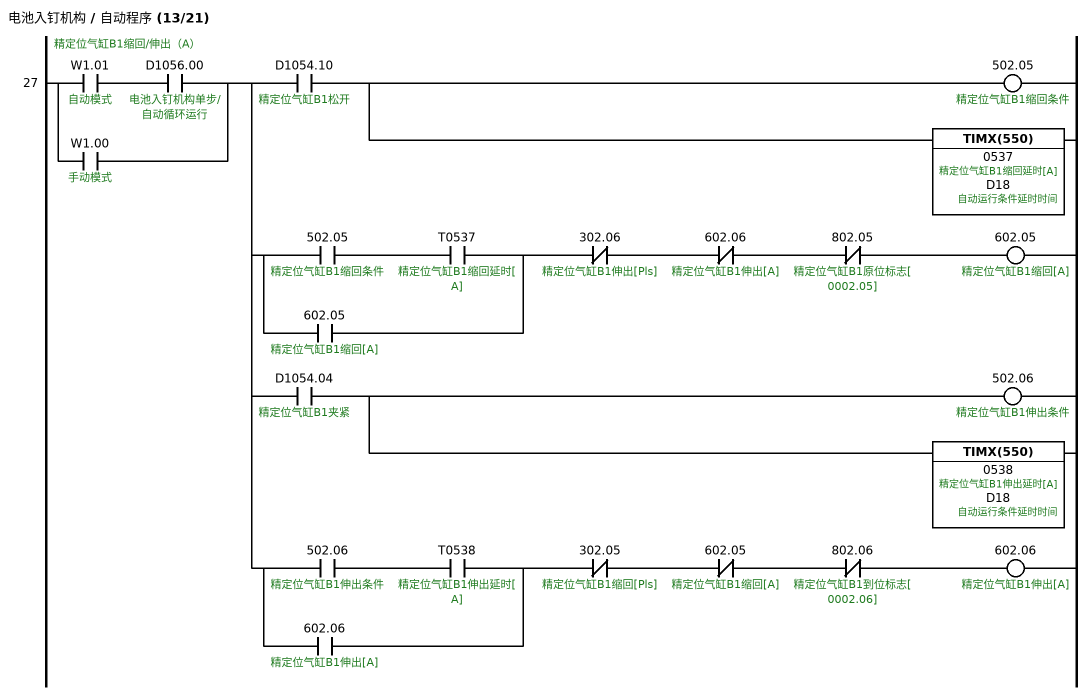
; rung 27: 精定位气缸B1缩回/伸出（A）
LD W1.01  ; 自动模式
AND D1056.00  ; 电池入钉机构单步/自动循环运行
OR W1.00  ; 手动模式
OUT TR0
AND D1054.10  ; 精定位气缸B1松开
OUT 502.05  ; 精定位气缸B1缩回条件
TIMX(550) 0537 D18  ; 自动运行条件延时时间, 精定位气缸B1缩回延时[A]
LD TR0
LD 502.05  ; 精定位气缸B1缩回条件
AND T0537  ; 精定位气缸B1缩回延时[A]
OR 602.05  ; 精定位气缸B1缩回[A]
ANDLD
ANDNOT 302.06  ; 精定位气缸B1伸出[Pls]
ANDNOT 602.06  ; 精定位气缸B1伸出[A]
ANDNOT 802.05  ; 精定位气缸B1原位标志[0002.05]
OUT 602.05  ; 精定位气缸B1缩回[A]
LD TR0
AND D1054.04  ; 精定位气缸B1夹紧
OUT 502.06  ; 精定位气缸B1伸出条件
TIMX(550) 0538 D18  ; 自动运行条件延时时间, 精定位气缸B1伸出延时[A]
LD TR0
LD 502.06  ; 精定位气缸B1伸出条件
AND T0538  ; 精定位气缸B1伸出延时[A]
OR 602.06  ; 精定位气缸B1伸出[A]
ANDLD
ANDNOT 302.05  ; 精定位气缸B1缩回[Pls]
ANDNOT 602.05  ; 精定位气缸B1缩回[A]
ANDNOT 802.06  ; 精定位气缸B1到位标志[0002.06]
OUT 602.06  ; 精定位气缸B1伸出[A]

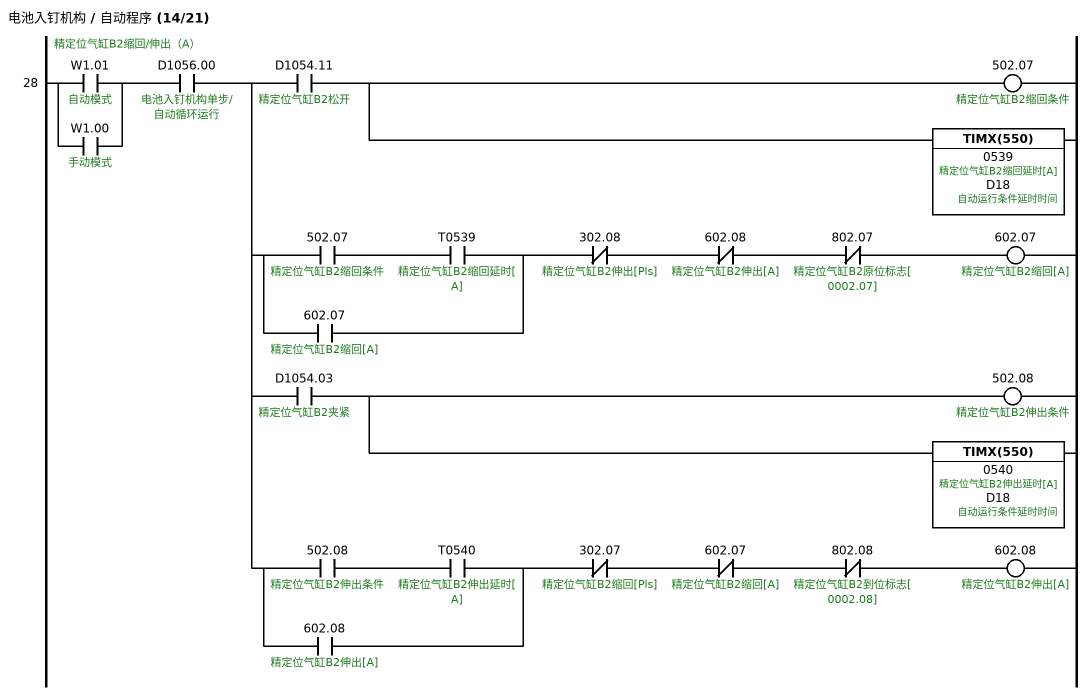
; rung 28: 精定位气缸B2缩回/伸出（A）
LD W1.01  ; 自动模式
OR W1.00  ; 手动模式
AND D1056.00  ; 电池入钉机构单步/自动循环运行
OUT TR0
AND D1054.11  ; 精定位气缸B2松开
OUT 502.07  ; 精定位气缸B2缩回条件
TIMX(550) 0539 D18  ; 自动运行条件延时时间, 精定位气缸B2缩回延时[A]
LD TR0
LD 502.07  ; 精定位气缸B2缩回条件
AND T0539  ; 精定位气缸B2缩回延时[A]
OR 602.07  ; 精定位气缸B2缩回[A]
ANDLD
ANDNOT 302.08  ; 精定位气缸B2伸出[Pls]
ANDNOT 602.08  ; 精定位气缸B2伸出[A]
ANDNOT 802.07  ; 精定位气缸B2原位标志[0002.07]
OUT 602.07  ; 精定位气缸B2缩回[A]
LD TR0
AND D1054.03  ; 精定位气缸B2夹紧
OUT 502.08  ; 精定位气缸B2伸出条件
TIMX(550) 0540 D18  ; 自动运行条件延时时间, 精定位气缸B2伸出延时[A]
LD TR0
LD 502.08  ; 精定位气缸B2伸出条件
AND T0540  ; 精定位气缸B2伸出延时[A]
OR 602.08  ; 精定位气缸B2伸出[A]
ANDLD
ANDNOT 302.07  ; 精定位气缸B2缩回[Pls]
ANDNOT 602.07  ; 精定位气缸B2缩回[A]
ANDNOT 802.08  ; 精定位气缸B2到位标志[0002.08]
OUT 602.08  ; 精定位气缸B2伸出[A]

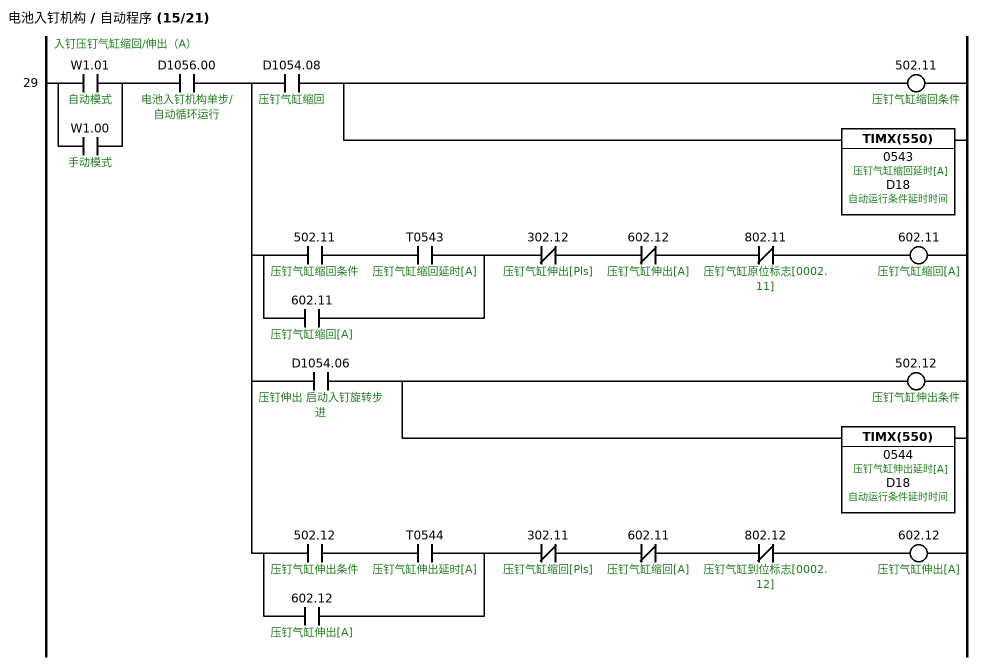
; rung 29: 入钉压钉气缸缩回/伸出（A）
LD W1.01  ; 自动模式
OR W1.00  ; 手动模式
AND D1056.00  ; 电池入钉机构单步/自动循环运行
OUT TR0
AND D1054.08  ; 压钉气缸缩回
OUT 502.11  ; 压钉气缸缩回条件
TIMX(550) 0543 D18  ; 自动运行条件延时时间, 压钉气缸缩回延时[A]
LD TR0
LD 502.11  ; 压钉气缸缩回条件
AND T0543  ; 压钉气缸缩回延时[A]
OR 602.11  ; 压钉气缸缩回[A]
ANDLD
ANDNOT 302.12  ; 压钉气缸伸出[Pls]
ANDNOT 602.12  ; 压钉气缸伸出[A]
ANDNOT 802.11  ; 压钉气缸原位标志[0002.11]
OUT 602.11  ; 压钉气缸缩回[A]
LD TR0
AND D1054.06  ; 压钉伸出 启动入钉旋转步进
OUT 502.12  ; 压钉气缸伸出条件
TIMX(550) 0544 D18  ; 自动运行条件延时时间, 压钉气缸伸出延时[A]
LD TR0
LD 502.12  ; 压钉气缸伸出条件
AND T0544  ; 压钉气缸伸出延时[A]
OR 602.12  ; 压钉气缸伸出[A]
ANDLD
ANDNOT 302.11  ; 压钉气缸缩回[Pls]
ANDNOT 602.11  ; 压钉气缸缩回[A]
ANDNOT 802.12  ; 压钉气缸到位标志[0002.12]
OUT 602.12  ; 压钉气缸伸出[A]

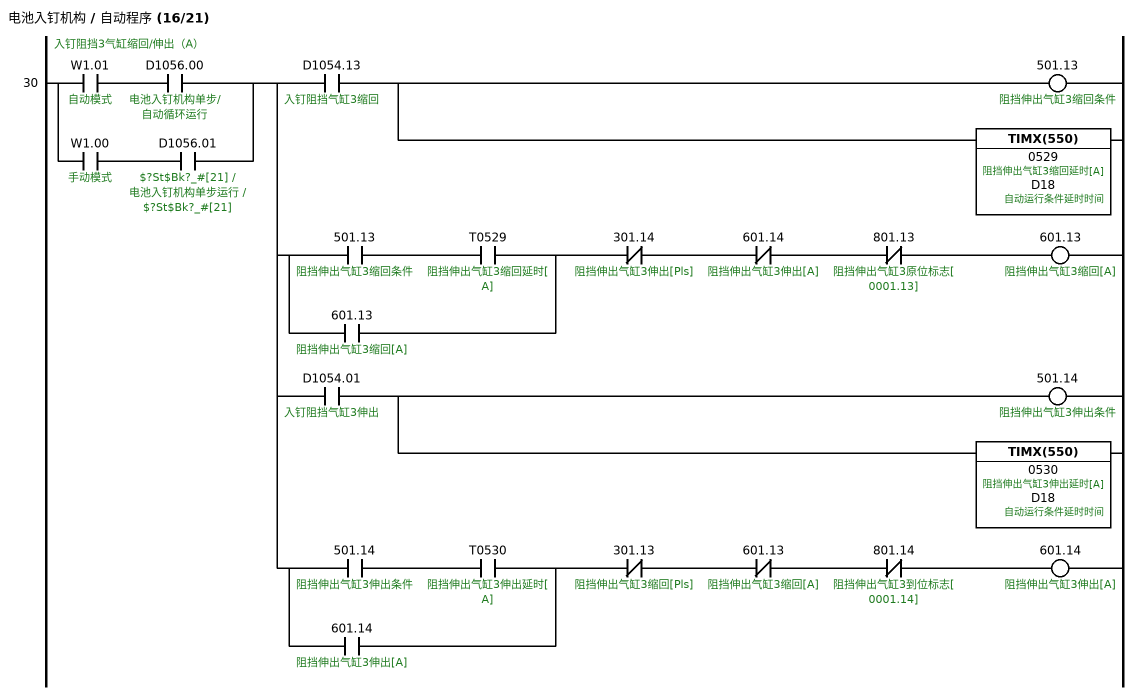
; rung 30: 入钉阻挡3气缸缩回/伸出（A）
LD W1.01  ; 自动模式
AND D1056.00  ; 电池入钉机构单步/自动循环运行
LD W1.00  ; 手动模式
AND D1056.01  ; $?St$Bk?_#[21] / 电池入钉机构单步运行 / $?St$Bk?_#[21]
ORLD
OUT TR0
AND D1054.13  ; 入钉阻挡气缸3缩回
OUT 501.13  ; 阻挡伸出气缸3缩回条件
TIMX(550) 0529 D18  ; 自动运行条件延时时间, 阻挡伸出气缸3缩回延时[A]
LD TR0
LD 501.13  ; 阻挡伸出气缸3缩回条件
AND T0529  ; 阻挡伸出气缸3缩回延时[A]
OR 601.13  ; 阻挡伸出气缸3缩回[A]
ANDLD
ANDNOT 301.14  ; 阻挡伸出气缸3伸出[Pls]
ANDNOT 601.14  ; 阻挡伸出气缸3伸出[A]
ANDNOT 801.13  ; 阻挡伸出气缸3原位标志[0001.13]
OUT 601.13  ; 阻挡伸出气缸3缩回[A]
LD TR0
AND D1054.01  ; 入钉阻挡气缸3伸出
OUT 501.14  ; 阻挡伸出气缸3伸出条件
TIMX(550) 0530 D18  ; 自动运行条件延时时间, 阻挡伸出气缸3伸出延时[A]
LD TR0
LD 501.14  ; 阻挡伸出气缸3伸出条件
AND T0530  ; 阻挡伸出气缸3伸出延时[A]
OR 601.14  ; 阻挡伸出气缸3伸出[A]
ANDLD
ANDNOT 301.13  ; 阻挡伸出气缸3缩回[Pls]
ANDNOT 601.13  ; 阻挡伸出气缸3缩回[A]
ANDNOT 801.14  ; 阻挡伸出气缸3到位标志[0001.14]
OUT 601.14  ; 阻挡伸出气缸3伸出[A]

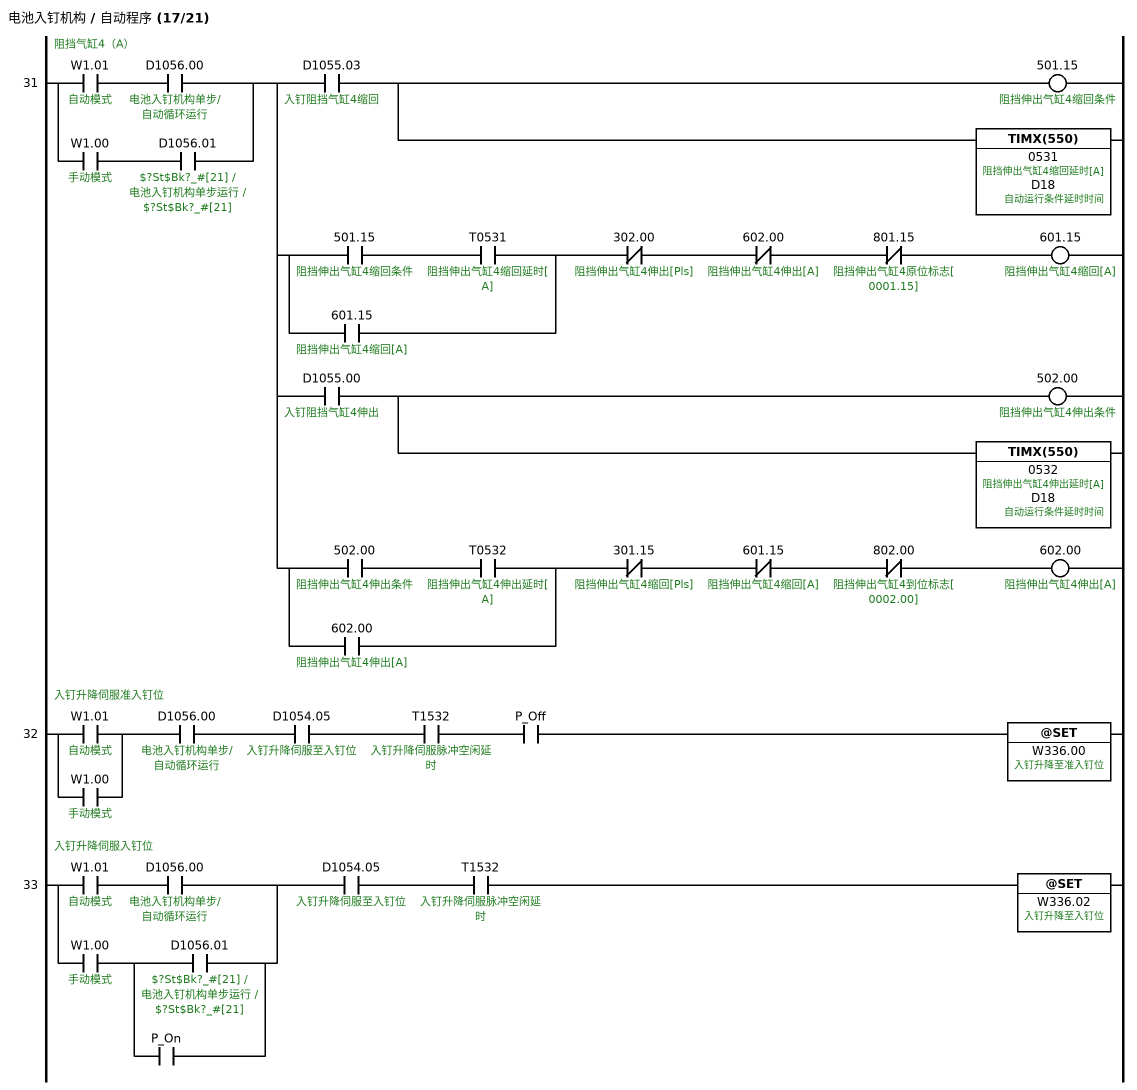
; rung 31: 阻挡气缸4（A）
LD W1.01  ; 自动模式
AND D1056.00  ; 电池入钉机构单步/自动循环运行
LD W1.00  ; 手动模式
AND D1056.01  ; $?St$Bk?_#[21] / 电池入钉机构单步运行 / $?St$Bk?_#[21]
ORLD
OUT TR0
AND D1055.03  ; 入钉阻挡气缸4缩回
OUT 501.15  ; 阻挡伸出气缸4缩回条件
TIMX(550) 0531 D18  ; 自动运行条件延时时间, 阻挡伸出气缸4缩回延时[A]
LD TR0
LD 501.15  ; 阻挡伸出气缸4缩回条件
AND T0531  ; 阻挡伸出气缸4缩回延时[A]
OR 601.15  ; 阻挡伸出气缸4缩回[A]
ANDLD
ANDNOT 302.00  ; 阻挡伸出气缸4伸出[Pls]
ANDNOT 602.00  ; 阻挡伸出气缸4伸出[A]
ANDNOT 801.15  ; 阻挡伸出气缸4原位标志[0001.15]
OUT 601.15  ; 阻挡伸出气缸4缩回[A]
LD TR0
AND D1055.00  ; 入钉阻挡气缸4伸出
OUT 502.00  ; 阻挡伸出气缸4伸出条件
TIMX(550) 0532 D18  ; 自动运行条件延时时间, 阻挡伸出气缸4伸出延时[A]
LD TR0
LD 502.00  ; 阻挡伸出气缸4伸出条件
AND T0532  ; 阻挡伸出气缸4伸出延时[A]
OR 602.00  ; 阻挡伸出气缸4伸出[A]
ANDLD
ANDNOT 301.15  ; 阻挡伸出气缸4缩回[Pls]
ANDNOT 601.15  ; 阻挡伸出气缸4缩回[A]
ANDNOT 802.00  ; 阻挡伸出气缸4到位标志[0002.00]
OUT 602.00  ; 阻挡伸出气缸4伸出[A]
; rung 32: 入钉升降伺服准入钉位
LD W1.01  ; 自动模式
OR W1.00  ; 手动模式
AND D1056.00  ; 电池入钉机构单步/自动循环运行
AND D1054.05  ; 入钉升降伺服至入钉位
AND T1532  ; 入钉升降伺服脉冲空闲延时
AND P_Off
@SET W336.00  ; 入钉升降至准入钉位
; rung 33: 入钉升降伺服入钉位
LD W1.01  ; 自动模式
AND D1056.00  ; 电池入钉机构单步/自动循环运行
LD W1.00  ; 手动模式
LD D1056.01  ; $?St$Bk?_#[21] / 电池入钉机构单步运行 / $?St$Bk?_#[21]
OR P_On
ANDLD
ORLD
AND D1054.05  ; 入钉升降伺服至入钉位
AND T1532  ; 入钉升降伺服脉冲空闲延时
@SET W336.02  ; 入钉升降至入钉位

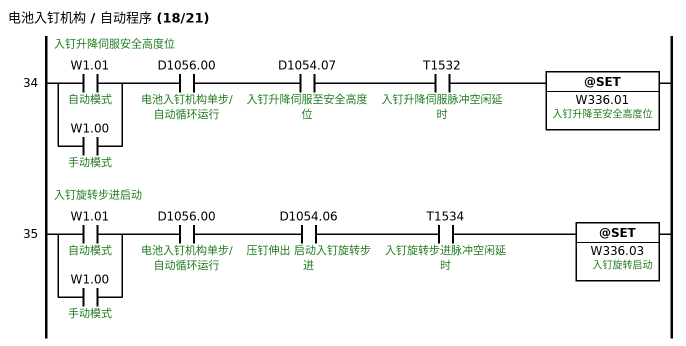
; rung 34: 入钉升降伺服安全高度位
LD W1.01  ; 自动模式
OR W1.00  ; 手动模式
AND D1056.00  ; 电池入钉机构单步/自动循环运行
AND D1054.07  ; 入钉升降伺服至安全高度位
AND T1532  ; 入钉升降伺服脉冲空闲延时
@SET W336.01  ; 入钉升降至安全高度位
; rung 35: 入钉旋转步进启动
LD W1.01  ; 自动模式
OR W1.00  ; 手动模式
AND D1056.00  ; 电池入钉机构单步/自动循环运行
AND D1054.06  ; 压钉伸出 启动入钉旋转步进
AND T1534  ; 入钉旋转步进脉冲空闲延时
@SET W336.03  ; 入钉旋转启动

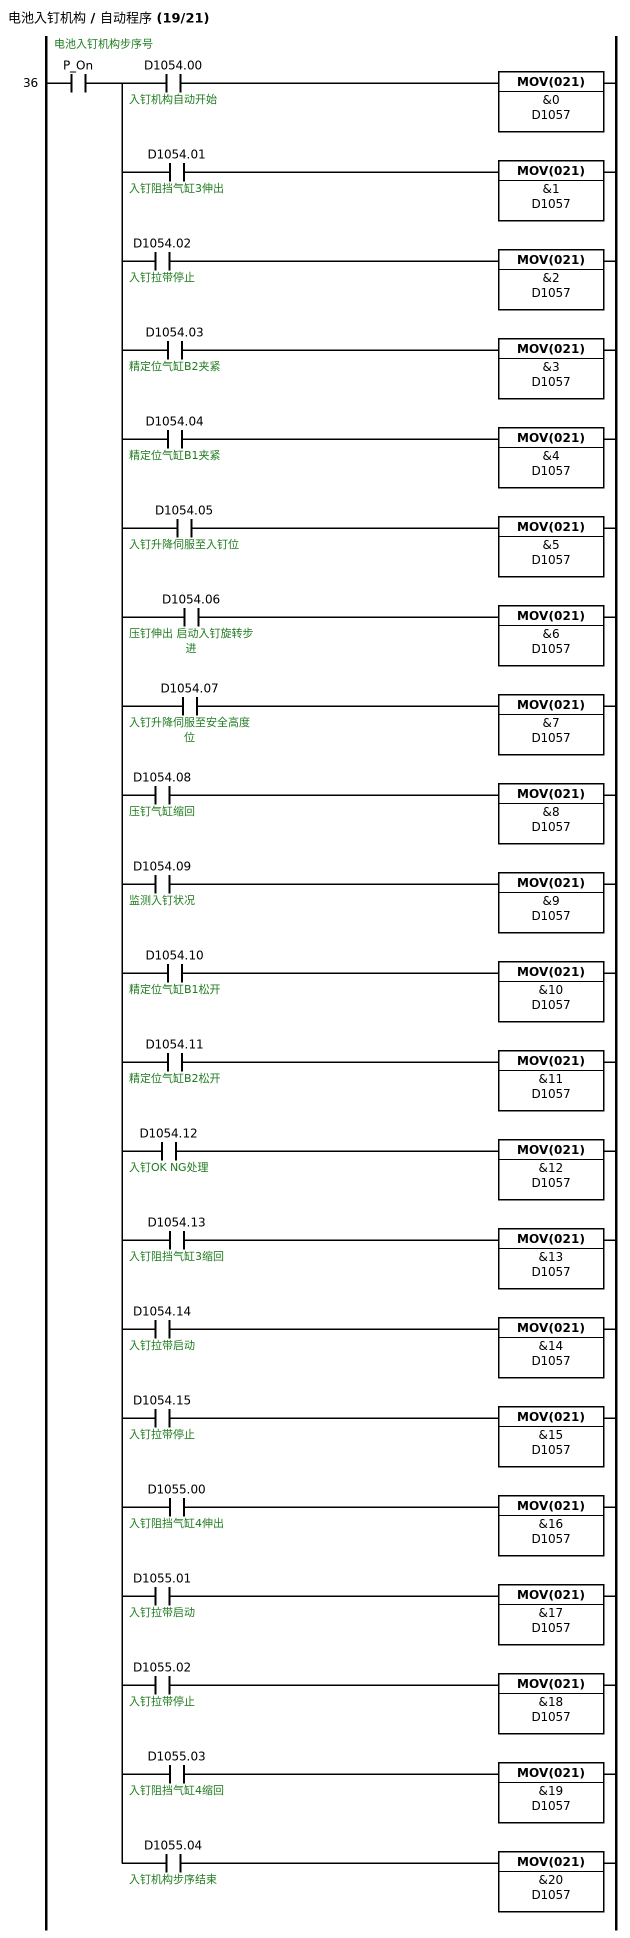
; rung 36: 电池入钉机构步序号
LD P_On
OUT TR0
AND D1054.00  ; 入钉机构自动开始
MOV(021) &0 D1057
LD TR0
AND D1054.01  ; 入钉阻挡气缸3伸出
MOV(021) &1 D1057
LD TR0
AND D1054.02  ; 入钉拉带停止
MOV(021) &2 D1057
LD TR0
AND D1054.03  ; 精定位气缸B2夹紧
MOV(021) &3 D1057
LD TR0
AND D1054.04  ; 精定位气缸B1夹紧
MOV(021) &4 D1057
LD TR0
AND D1054.05  ; 入钉升降伺服至入钉位
MOV(021) &5 D1057
LD TR0
AND D1054.06  ; 压钉伸出 启动入钉旋转步进
MOV(021) &6 D1057
LD TR0
AND D1054.07  ; 入钉升降伺服至安全高度位
MOV(021) &7 D1057
LD TR0
AND D1054.08  ; 压钉气缸缩回
MOV(021) &8 D1057
LD TR0
AND D1054.09  ; 监测入钉状况
MOV(021) &9 D1057
LD TR0
AND D1054.10  ; 精定位气缸B1松开
MOV(021) &10 D1057
LD TR0
AND D1054.11  ; 精定位气缸B2松开
MOV(021) &11 D1057
LD TR0
AND D1054.12  ; 入钉OK NG处理
MOV(021) &12 D1057
LD TR0
AND D1054.13  ; 入钉阻挡气缸3缩回
MOV(021) &13 D1057
LD TR0
AND D1054.14  ; 入钉拉带启动
MOV(021) &14 D1057
LD TR0
AND D1054.15  ; 入钉拉带停止
MOV(021) &15 D1057
LD TR0
AND D1055.00  ; 入钉阻挡气缸4伸出
MOV(021) &16 D1057
LD TR0
AND D1055.01  ; 入钉拉带启动
MOV(021) &17 D1057
LD TR0
AND D1055.02  ; 入钉拉带停止
MOV(021) &18 D1057
LD TR0
AND D1055.03  ; 入钉阻挡气缸4缩回
MOV(021) &19 D1057
LD TR0
AND D1055.04  ; 入钉机构步序结束
MOV(021) &20 D1057

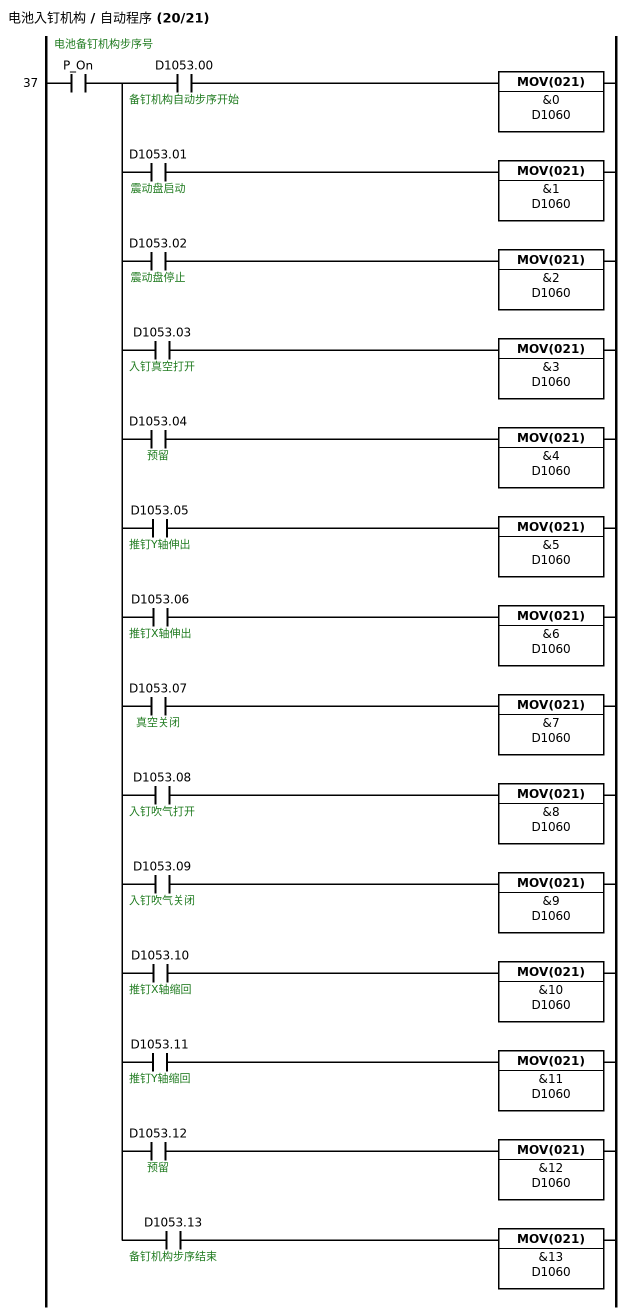
; rung 37: 电池备钉机构步序号
LD P_On
OUT TR0
AND D1053.00  ; 备钉机构自动步序开始
MOV(021) &0 D1060
LD TR0
AND D1053.01  ; 震动盘启动
MOV(021) &1 D1060
LD TR0
AND D1053.02  ; 震动盘停止
MOV(021) &2 D1060
LD TR0
AND D1053.03  ; 入钉真空打开
MOV(021) &3 D1060
LD TR0
AND D1053.04  ; 预留
MOV(021) &4 D1060
LD TR0
AND D1053.05  ; 推钉Y轴伸出
MOV(021) &5 D1060
LD TR0
AND D1053.06  ; 推钉X轴伸出
MOV(021) &6 D1060
LD TR0
AND D1053.07  ; 真空关闭
MOV(021) &7 D1060
LD TR0
AND D1053.08  ; 入钉吹气打开
MOV(021) &8 D1060
LD TR0
AND D1053.09  ; 入钉吹气关闭
MOV(021) &9 D1060
LD TR0
AND D1053.10  ; 推钉X轴缩回
MOV(021) &10 D1060
LD TR0
AND D1053.11  ; 推钉Y轴缩回
MOV(021) &11 D1060
LD TR0
AND D1053.12  ; 预留
MOV(021) &12 D1060
LD TR0
AND D1053.13  ; 备钉机构步序结束
MOV(021) &13 D1060

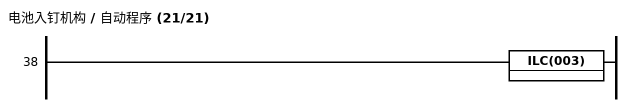
; rung 38
ILC(003)

### Section 状态指示灯

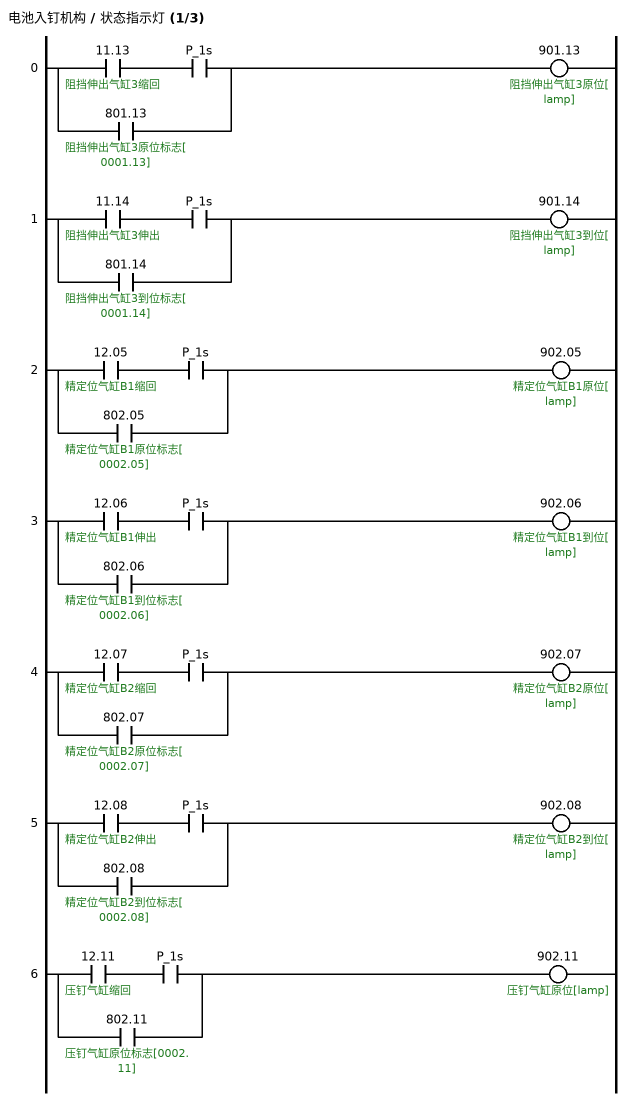
; rung 0
LD 11.13  ; 阻挡伸出气缸3缩回
AND P_1s
OR 801.13  ; 阻挡伸出气缸3原位标志[0001.13]
OUT 901.13  ; 阻挡伸出气缸3原位[lamp]
; rung 1
LD 11.14  ; 阻挡伸出气缸3伸出
AND P_1s
OR 801.14  ; 阻挡伸出气缸3到位标志[0001.14]
OUT 901.14  ; 阻挡伸出气缸3到位[lamp]
; rung 2
LD 12.05  ; 精定位气缸B1缩回
AND P_1s
OR 802.05  ; 精定位气缸B1原位标志[0002.05]
OUT 902.05  ; 精定位气缸B1原位[lamp]
; rung 3
LD 12.06  ; 精定位气缸B1伸出
AND P_1s
OR 802.06  ; 精定位气缸B1到位标志[0002.06]
OUT 902.06  ; 精定位气缸B1到位[lamp]
; rung 4
LD 12.07  ; 精定位气缸B2缩回
AND P_1s
OR 802.07  ; 精定位气缸B2原位标志[0002.07]
OUT 902.07  ; 精定位气缸B2原位[lamp]
; rung 5
LD 12.08  ; 精定位气缸B2伸出
AND P_1s
OR 802.08  ; 精定位气缸B2到位标志[0002.08]
OUT 902.08  ; 精定位气缸B2到位[lamp]
; rung 6
LD 12.11  ; 压钉气缸缩回
AND P_1s
OR 802.11  ; 压钉气缸原位标志[0002.11]
OUT 902.11  ; 压钉气缸原位[lamp]

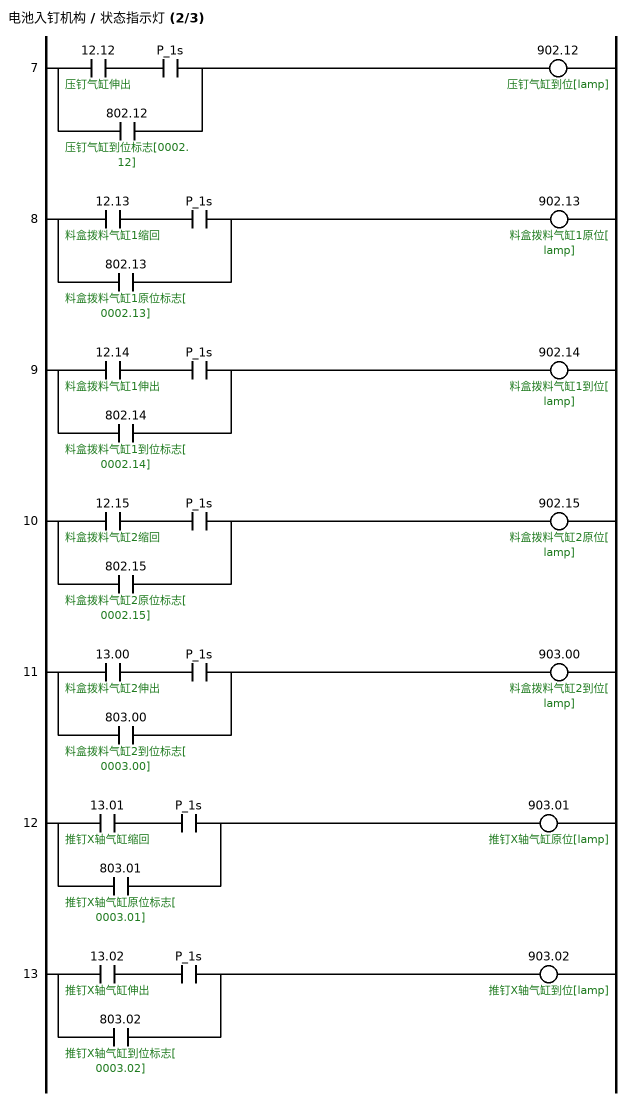
; rung 7
LD 12.12  ; 压钉气缸伸出
AND P_1s
OR 802.12  ; 压钉气缸到位标志[0002.12]
OUT 902.12  ; 压钉气缸到位[lamp]
; rung 8
LD 12.13  ; 料盒拨料气缸1缩回
AND P_1s
OR 802.13  ; 料盒拨料气缸1原位标志[0002.13]
OUT 902.13  ; 料盒拨料气缸1原位[lamp]
; rung 9
LD 12.14  ; 料盒拨料气缸1伸出
AND P_1s
OR 802.14  ; 料盒拨料气缸1到位标志[0002.14]
OUT 902.14  ; 料盒拨料气缸1到位[lamp]
; rung 10
LD 12.15  ; 料盒拨料气缸2缩回
AND P_1s
OR 802.15  ; 料盒拨料气缸2原位标志[0002.15]
OUT 902.15  ; 料盒拨料气缸2原位[lamp]
; rung 11
LD 13.00  ; 料盒拨料气缸2伸出
AND P_1s
OR 803.00  ; 料盒拨料气缸2到位标志[0003.00]
OUT 903.00  ; 料盒拨料气缸2到位[lamp]
; rung 12
LD 13.01  ; 推钉X轴气缸缩回
AND P_1s
OR 803.01  ; 推钉X轴气缸原位标志[0003.01]
OUT 903.01  ; 推钉X轴气缸原位[lamp]
; rung 13
LD 13.02  ; 推钉X轴气缸伸出
AND P_1s
OR 803.02  ; 推钉X轴气缸到位标志[0003.02]
OUT 903.02  ; 推钉X轴气缸到位[lamp]

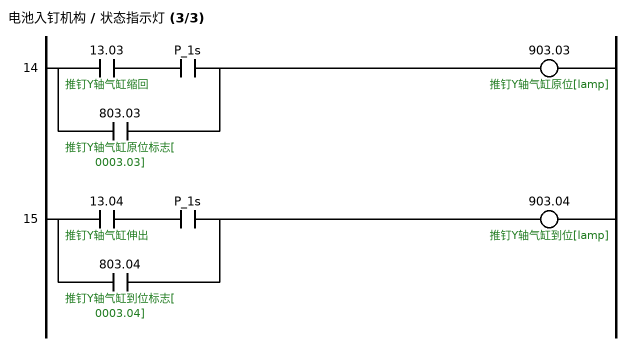
; rung 14
LD 13.03  ; 推钉Y轴气缸缩回
AND P_1s
OR 803.03  ; 推钉Y轴气缸原位标志[0003.03]
OUT 903.03  ; 推钉Y轴气缸原位[lamp]
; rung 15
LD 13.04  ; 推钉Y轴气缸伸出
AND P_1s
OR 803.04  ; 推钉Y轴气缸到位标志[0003.04]
OUT 903.04  ; 推钉Y轴气缸到位[lamp]

### Section 输出程序

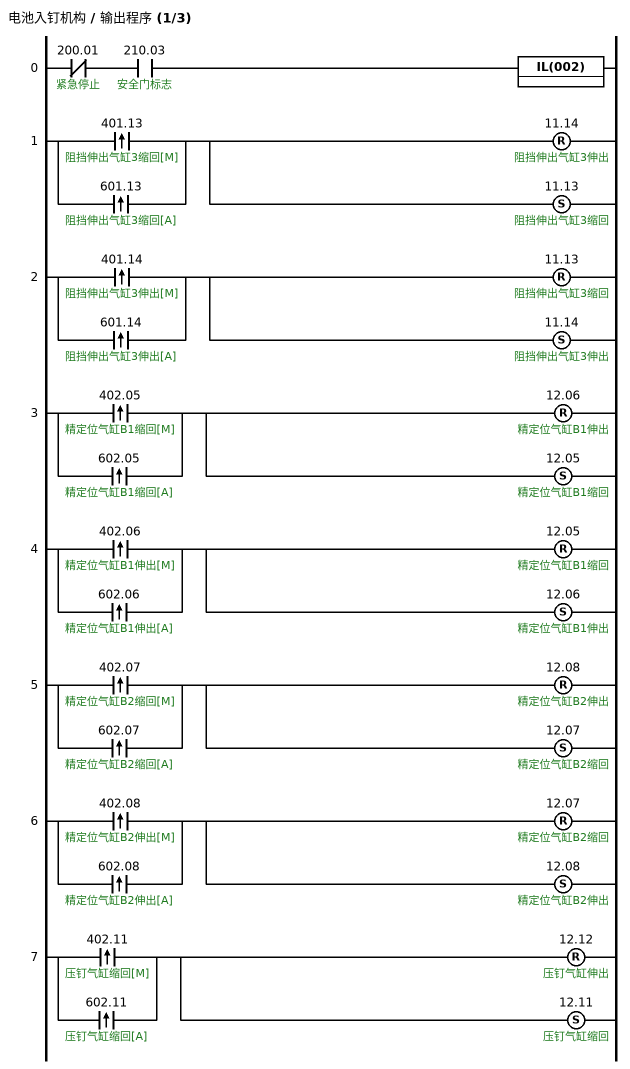
; rung 0
LDNOT 200.01  ; 紧急停止
AND 210.03  ; 安全门标志
IL(002)
; rung 1
@LD 401.13  ; 阻挡伸出气缸3缩回[M]
@OR 601.13  ; 阻挡伸出气缸3缩回[A]
RSET 11.14  ; 阻挡伸出气缸3伸出
SET 11.13  ; 阻挡伸出气缸3缩回
; rung 2
@LD 401.14  ; 阻挡伸出气缸3伸出[M]
@OR 601.14  ; 阻挡伸出气缸3伸出[A]
RSET 11.13  ; 阻挡伸出气缸3缩回
SET 11.14  ; 阻挡伸出气缸3伸出
; rung 3
@LD 402.05  ; 精定位气缸B1缩回[M]
@OR 602.05  ; 精定位气缸B1缩回[A]
RSET 12.06  ; 精定位气缸B1伸出
SET 12.05  ; 精定位气缸B1缩回
; rung 4
@LD 402.06  ; 精定位气缸B1伸出[M]
@OR 602.06  ; 精定位气缸B1伸出[A]
RSET 12.05  ; 精定位气缸B1缩回
SET 12.06  ; 精定位气缸B1伸出
; rung 5
@LD 402.07  ; 精定位气缸B2缩回[M]
@OR 602.07  ; 精定位气缸B2缩回[A]
RSET 12.08  ; 精定位气缸B2伸出
SET 12.07  ; 精定位气缸B2缩回
; rung 6
@LD 402.08  ; 精定位气缸B2伸出[M]
@OR 602.08  ; 精定位气缸B2伸出[A]
RSET 12.07  ; 精定位气缸B2缩回
SET 12.08  ; 精定位气缸B2伸出
; rung 7
@LD 402.11  ; 压钉气缸缩回[M]
@OR 602.11  ; 压钉气缸缩回[A]
RSET 12.12  ; 压钉气缸伸出
SET 12.11  ; 压钉气缸缩回

